LIN {X 0,Y 500.021,Z 595.129,A -85,B 0,C 180,E1 -13691.31,E2 -13691.31} C_VEL
LIN {X 0,Y 499.964,Z 595.135,A -85,B 0,C 180,E1 -13694.832,E2 -13694.832} C_VEL
LIN {X 0,Y 499.873,Z 595.155,A -85,B 0,C 180,E1 -13697.955,E2 -13697.955} C_VEL
LIN {X 0,Y 499.868,Z 595.149,A -85,B 0,C 180,E1 -13700.507,E2 -13700.507} C_VEL
LIN {X 0,Y 499.856,Z 595.149,A -85,B 0,C 180,E1 -13703.102,E2 -13703.102} C_VEL
LIN {X 0,Y 499.832,Z 595.157,A -85,B 0,C 180,E1 -13705.749,E2 -13705.749} C_VEL
LIN {X 0,Y 499.854,Z 595.151,A -85,B 0,C 180,E1 -13708.453,E2 -13708.453} C_VEL
LIN {X 0,Y 499.831,Z 595.152,A -85,B 0,C 180,E1 -13711.259,E2 -13711.259} C_VEL
LIN {X 0,Y 499.847,Z 595.155,A -85,B 0,C 180,E1 -13714.231,E2 -13714.231} C_VEL
LIN {X 0,Y 499.88,Z 595.146,A -85,B 0,C 180,E1 -13717.051,E2 -13717.051} C_VEL
LIN {X 0,Y 499.824,Z 595.159,A -85,B 0,C 180,E1 -13720.138,E2 -13720.138} C_VEL
LIN {X 0,Y 499.878,Z 595.147,A -85,B 0,C 180,E1 -13723.362,E2 -13723.362} C_VEL
LIN {X 0,Y 499.877,Z 595.146,A -85,B 0,C 180,E1 -13726.773,E2 -13726.773} C_VEL
LIN {X 0,Y 499.823,Z 595.16,A -85,B 0,C 180,E1 -13729.862,E2 -13729.862} C_VEL
LIN {X 0,Y 499.832,Z 595.151,A -85,B 0,C 180,E1 -13733.013,E2 -13733.013} C_VEL
LIN {X 0,Y 499.84,Z 595.158,A -85,B 0,C 180,E1 -13735.907,E2 -13735.907} C_VEL
LIN {X 0,Y 499.835,Z 595.152,A -85,B 0,C 180,E1 -13738.768,E2 -13738.768} C_VEL
LIN {X 0,Y 499.834,Z 595.154,A -85,B 0,C 180,E1 -13741.546,E2 -13741.546} C_VEL
LIN {X 0,Y 499.832,Z 595.16,A -85,B 0,C 180,E1 -13744.252,E2 -13744.252} C_VEL
LIN {X 0,Y 499.914,Z 595.236,A -85,B 0,C 180,E1 -13745.236,E2 -13745.236} C_VEL
LIN {X 0,Y 502.292,Z 608.896,A -85,B 0,C 180,E1 -13747.882,E2 -13747.882} C_VEL
LIN {X 0,Y 501.344,Z 623.933,A -85,B 0,C 180,E1 -13750.621,E2 -13750.621} C_VEL
LIN {X 0,Y 500.239,Z 642.384,A -85,B 0,C 180,E1 -13753.946,E2 -13753.946} C_VEL
LIN {X 0,Y 500.096,Z 646.425,A -85,B 0,C 180,E1 -13754.636,E2 -13754.636} C_VEL
LIN {X 0,Y 503.159,Z 673.816,A -85,B 0,C 180,E1 -13755.185,E2 -13755.185} C_VEL
LIN {X 0,Y 501.946,Z 752.433,A -85,B 0,C 180,E1 -13756.534,E2 -13756.534} C_VEL
LIN {X 0,Y 501.731,Z 762.36,A -85,B 0,C 180,E1 -13756.785,E2 -13756.785} C_VEL
LIN {X 0,Y 501.395,Z 772.419,A -85,B 0,C 180,E1 -13757.136,E2 -13757.136} C_VEL
LIN {X 0,Y 501.08,Z 782.406,A -85,B 0,C 180,E1 -13757.589,E2 -13757.589} C_VEL
LIN {X 0,Y 500.684,Z 792.552,A -85,B 0,C 180,E1 -13758.17,E2 -13758.17} C_VEL
LIN {X 0,Y 500.217,Z 802.826,A -85,B 0,C 180,E1 -13758.899,E2 -13758.899} C_VEL
LIN {X 0,Y 499.783,Z 811.123,A -85,B 0,C 180,E1 -13759.605,E2 -13759.605} C_VEL
LIN {X 0,Y 499.348,Z 820.005,A -85,B 0,C 180,E1 -13760.513,E2 -13760.513} C_VEL
LIN {X 0,Y 498.984,Z 826.725,A -85,B 0,C 180,E1 -13761.321,E2 -13761.321} C_VEL
LIN {X 0,Y 498.712,Z 833.772,A -85,B 0,C 180,E1 -13762.332,E2 -13762.332} C_VEL
LIN {X 0,Y 498.462,Z 840.635,A -85,B 0,C 180,E1 -13763.545,E2 -13763.545} C_VEL
LIN {X 0,Y 498.34,Z 844.527,A -85,B 0,C 180,E1 -13764.354,E2 -13764.354} C_VEL
LIN {X 0,Y 498.199,Z 849.173,A -85,B 0,C 180,E1 -13765.565,E2 -13765.565} C_VEL
LIN {X 0,Y 498.143,Z 852.679,A -85,B 0,C 180,E1 -13766.776,E2 -13766.776} C_VEL
LIN {X 0,Y 498.16,Z 855.649,A -85,B 0,C 180,E1 -13768.389,E2 -13768.389} C_VEL
LIN {X 0,Y 498.171,Z 856.61,A -85,B 0,C 180,E1 -13769.195,E2 -13769.195} C_VEL
LIN {X 0,Y 498.15,Z 857.003,A -85,B 0,C 180,E1 -13770.806,E2 -13770.806} C_VEL
LIN {X 0,Y 498.124,Z 856.638,A -85,B 0,C 180,E1 -13771.612,E2 -13771.612} C_VEL
LIN {X 0,Y 498.144,Z 854.362,A -85,B 0,C 180,E1 -13773.306,E2 -13773.306} C_VEL
LIN {X 0,Y 498.201,Z 851.826,A -85,B 0,C 180,E1 -13774.435,E2 -13774.435} C_VEL
LIN {X 0,Y 498.384,Z 848.053,A -85,B 0,C 180,E1 -13775.646,E2 -13775.646} C_VEL
LIN {X 0,Y 498.634,Z 843.12,A -85,B 0,C 180,E1 -13776.858,E2 -13776.858} C_VEL
LIN {X 0,Y 499.019,Z 836.872,A -85,B 0,C 180,E1 -13778.069,E2 -13778.069} C_VEL
LIN {X 0,Y 499.423,Z 830.563,A -85,B 0,C 180,E1 -13779.078,E2 -13779.078} C_VEL
LIN {X 0,Y 500.017,Z 822.995,A -85,B 0,C 180,E1 -13780.085,E2 -13780.085} C_VEL
LIN {X 0,Y 500.639,Z 814.859,A -85,B 0,C 180,E1 -13780.99,E2 -13780.99} C_VEL
LIN {X 0,Y 501.277,Z 805.922,A -85,B 0,C 180,E1 -13781.82,E2 -13781.82} C_VEL
LIN {X 0,Y 501.901,Z 796.264,A -85,B 0,C 180,E1 -13782.565,E2 -13782.565} C_VEL
LIN {X 0,Y 502.454,Z 786.303,A -85,B 0,C 180,E1 -13783.196,E2 -13783.196} C_VEL
LIN {X 0,Y 503.002,Z 776.582,A -85,B 0,C 180,E1 -13783.694,E2 -13783.694} C_VEL
LIN {X 0,Y 503.622,Z 765.279,A -85,B 0,C 180,E1 -13784.138,E2 -13784.138} C_VEL
LIN {X 0,Y 504.029,Z 755.185,A -85,B 0,C 180,E1 -13784.435,E2 -13784.435} C_VEL
LIN {X 0,Y 504.455,Z 737.22,A -85,B 0,C 180,E1 -13784.782,E2 -13784.782} C_VEL
LIN {X 0,Y 505.705,Z 672.59,A -85,B 0,C 180,E1 -13785.956,E2 -13785.956} C_VEL
LIN {X 0,Y 503.052,Z 654.485,A -85,B 0,C 180,E1 -13786.438,E2 -13786.438} C_VEL
LIN {X 0,Y 501.115,Z 644.89,A -85,B 0,C 180,E1 -13786.724,E2 -13786.724} C_VEL
LIN {X 0,Y 502.421,Z 628.877,A -85,B 0,C 180,E1 -13789.76,E2 -13789.76} C_VEL
LIN {X 0,Y 503.702,Z 615.998,A -85,B 0,C 180,E1 -13792.268,E2 -13792.268} C_VEL
LIN {X 0,Y 503.047,Z 610.412,A -85,B 0,C 180,E1 -13793.467,E2 -13793.467} C_VEL
LIN {X 0,Y 501.107,Z 600.725,A -85,B 0,C 180,E1 -13795.678,E2 -13795.678} C_VEL
LIN {X 0,Y 499.876,Z 595.157,A -85,B 0,C 180,E1 -13797.035,E2 -13797.035} C_VEL
LIN {X 0,Y 499.844,Z 595.157,A -85,B 0,C 180,E1 -13800.297,E2 -13800.297} C_VEL
LIN {X 0,Y 499.851,Z 595.156,A -85,B 0,C 180,E1 -13803.128,E2 -13803.128} C_VEL
LIN {X 0,Y 499.902,Z 595.145,A -85,B 0,C 180,E1 -13806.05,E2 -13806.05} C_VEL
LIN {X 0,Y 499.84,Z 595.151,A -85,B 0,C 180,E1 -13809.095,E2 -13809.095} C_VEL
LIN {X 0,Y 499.843,Z 595.15,A -85,B 0,C 180,E1 -13812.271,E2 -13812.271} C_VEL
LIN {X 0,Y 499.883,Z 595.148,A -85,B 0,C 180,E1 -13814.476,E2 -13814.476} C_VEL
LIN {X 0,Y 499.858,Z 595.154,A -85,B 0,C 180,E1 -13817.731,E2 -13817.731} C_VEL
LIN {X 0,Y 499.895,Z 595.148,A -85,B 0,C 180,E1 -13820.413,E2 -13820.413} C_VEL
LIN {X 0,Y 499.908,Z 595.145,A -85,B 0,C 180,E1 -13823.951,E2 -13823.951} C_VEL
LIN {X 0,Y 499.9,Z 595.149,A -85,B 0,C 180,E1 -13827.215,E2 -13827.215} C_VEL
LIN {X 0,Y 499.889,Z 595.148,A -85,B 0,C 180,E1 -13830.313,E2 -13830.313} C_VEL
LIN {X 0,Y 499.884,Z 595.151,A -85,B 0,C 180,E1 -13833.36,E2 -13833.36} C_VEL
LIN {X 0,Y 499.88,Z 595.15,A -85,B 0,C 180,E1 -13836.024,E2 -13836.024} C_VEL
LIN {X 0,Y 499.921,Z 595.151,A -85,B 0,C 180,E1 -13838.636,E2 -13838.636} C_VEL
LIN {X 0,Y 499.892,Z 595.155,A -85,B 0,C 180,E1 -13841.199,E2 -13841.199} C_VEL
LIN {X 0,Y 499.902,Z 595.151,A -85,B 0,C 180,E1 -13843.726,E2 -13843.726} C_VEL
LIN {X 0,Y 499.988,Z 595.223,A -85,B 0,C 180,E1 -13845.964,E2 -13845.964} C_VEL
LIN {X 0,Y 502.17,Z 605.861,A -85,B 0,C 180,E1 -13848.739,E2 -13848.739} C_VEL
LIN {X 0,Y 502.914,Z 610.897,A -85,B 0,C 180,E1 -13849.974,E2 -13849.974} C_VEL
LIN {X 0,Y 502.468,Z 618.166,A -85,B 0,C 180,E1 -13851.623,E2 -13851.623} C_VEL
LIN {X 0,Y 501.77,Z 626.142,A -85,B 0,C 180,E1 -13853.361,E2 -13853.361} C_VEL
LIN {X 0,Y 505.297,Z 642.925,A -85,B 0,C 180,E1 -13853.87,E2 -13853.87} C_VEL
LIN {X 0,Y 506.244,Z 649.346,A -85,B 0,C 180,E1 -13854.043,E2 -13854.043} C_VEL
LIN {X 0,Y 504.557,Z 711.904,A -85,B 0,C 180,E1 -13855.172,E2 -13855.172} C_VEL
LIN {X 0,Y 504.07,Z 733.839,A -85,B 0,C 180,E1 -13855.592,E2 -13855.592} C_VEL
LIN {X 0,Y 503.663,Z 745.565,A -85,B 0,C 180,E1 -13855.938,E2 -13855.938} C_VEL
LIN {X 0,Y 503.125,Z 759.1,A -85,B 0,C 180,E1 -13856.508,E2 -13856.508} C_VEL
LIN {X 0,Y 502.558,Z 771.102,A -85,B 0,C 180,E1 -13857.204,E2 -13857.204} C_VEL
LIN {X 0,Y 502.01,Z 780.801,A -85,B 0,C 180,E1 -13857.901,E2 -13857.901} C_VEL
LIN {X 0,Y 501.393,Z 789.985,A -85,B 0,C 180,E1 -13858.699,E2 -13858.699} C_VEL
LIN {X 0,Y 500.692,Z 798.607,A -85,B 0,C 180,E1 -13859.599,E2 -13859.599} C_VEL
LIN {X 0,Y 500.106,Z 805.153,A -85,B 0,C 180,E1 -13860.401,E2 -13860.401} C_VEL
LIN {X 0,Y 499.598,Z 812.014,A -85,B 0,C 180,E1 -13861.406,E2 -13861.406} C_VEL
LIN {X 0,Y 499.104,Z 817.772,A -85,B 0,C 180,E1 -13862.413,E2 -13862.413} C_VEL
LIN {X 0,Y 498.802,Z 823.337,A -85,B 0,C 180,E1 -13863.623,E2 -13863.623} C_VEL
LIN {X 0,Y 498.54,Z 827.721,A -85,B 0,C 180,E1 -13864.835,E2 -13864.835} C_VEL
LIN {X 0,Y 498.413,Z 830.206,A -85,B 0,C 180,E1 -13865.706,E2 -13865.706} C_VEL
LIN {X 0,Y 498.149,Z 833.293,A -85,B 0,C 180,E1 -13867.27,E2 -13867.27} C_VEL
LIN {X 0,Y 498.062,Z 834.271,A -85,B 0,C 180,E1 -13868.084,E2 -13868.084} C_VEL
LIN {X 0,Y 498.099,Z 834.913,A -85,B 0,C 180,E1 -13869.715,E2 -13869.715} C_VEL
LIN {X 0,Y 498.076,Z 834.546,A -85,B 0,C 180,E1 -13870.534,E2 -13870.534} C_VEL
LIN {X 0,Y 498.017,Z 832.61,A -85,B 0,C 180,E1 -13872.179,E2 -13872.179} C_VEL
LIN {X 0,Y 498.168,Z 829.923,A -85,B 0,C 180,E1 -13873.414,E2 -13873.414} C_VEL
LIN {X 0,Y 498.34,Z 826.113,A -85,B 0,C 180,E1 -13874.655,E2 -13874.655} C_VEL
LIN {X 0,Y 498.51,Z 821.045,A -85,B 0,C 180,E1 -13875.901,E2 -13875.901} C_VEL
LIN {X 0,Y 498.76,Z 815.812,A -85,B 0,C 180,E1 -13876.942,E2 -13876.942} C_VEL
LIN {X 0,Y 498.967,Z 809.412,A -85,B 0,C 180,E1 -13877.989,E2 -13877.989} C_VEL
LIN {X 0,Y 499.369,Z 801.644,A -85,B 0,C 180,E1 -13879.033,E2 -13879.033} C_VEL
LIN {X 0,Y 499.785,Z 792.659,A -85,B 0,C 180,E1 -13880.028,E2 -13880.028} C_VEL
LIN {X 0,Y 500.124,Z 784.129,A -85,B 0,C 180,E1 -13880.817,E2 -13880.817} C_VEL
LIN {X 0,Y 500.617,Z 774.605,A -85,B 0,C 180,E1 -13881.548,E2 -13881.548} C_VEL
LIN {X 0,Y 501.03,Z 764.623,A -85,B 0,C 180,E1 -13882.176,E2 -13882.176} C_VEL
LIN {X 0,Y 501.379,Z 754.57,A -85,B 0,C 180,E1 -13882.687,E2 -13882.687} C_VEL
LIN {X 0,Y 501.611,Z 743.432,A -85,B 0,C 180,E1 -13883.124,E2 -13883.124} C_VEL
LIN {X 0,Y 501.903,Z 732.354,A -85,B 0,C 180,E1 -13883.437,E2 -13883.437} C_VEL
LIN {X 0,Y 502.427,Z 709.429,A -85,B 0,C 180,E1 -13883.847,E2 -13883.847} C_VEL
LIN {X 0,Y 503.284,Z 645.821,A -85,B 0,C 180,E1 -13884.934,E2 -13884.934} C_VEL
LIN {X 0,Y 500.222,Z 624.306,A -85,B 0,C 180,E1 -13885.398,E2 -13885.398} C_VEL
LIN {X 0,Y 501.029,Z 609.69,A -85,B 0,C 180,E1 -13888.38,E2 -13888.38} C_VEL
LIN {X 0,Y 501.279,Z 603.782,A -85,B 0,C 180,E1 -13889.603,E2 -13889.603} C_VEL
LIN {X 0,Y 499.955,Z 595.145,A -85,B 0,C 180,E1 -13891.488,E2 -13891.488} C_VEL
LIN {X 0,Y 499.881,Z 595.15,A -85,B 0,C 180,E1 -13894.236,E2 -13894.236} C_VEL
LIN {X 0,Y 499.889,Z 595.144,A -85,B 0,C 180,E1 -13897.05,E2 -13897.05} C_VEL
LIN {X 0,Y 499.879,Z 595.152,A -85,B 0,C 180,E1 -13900.132,E2 -13900.132} C_VEL
LIN {X 0,Y 499.88,Z 595.147,A -85,B 0,C 180,E1 -13903.361,E2 -13903.361} C_VEL
LIN {X 0,Y 499.88,Z 595.146,A -85,B 0,C 180,E1 -13906.638,E2 -13906.638} C_VEL
LIN {X 0,Y 499.878,Z 595.153,A -85,B 0,C 180,E1 -13909.867,E2 -13909.867} C_VEL
LIN {X 0,Y 499.89,Z 595.144,A -85,B 0,C 180,E1 -13913.004,E2 -13913.004} C_VEL
LIN {X 0,Y 499.869,Z 595.155,A -85,B 0,C 180,E1 -13915.909,E2 -13915.909} C_VEL
LIN {X 0,Y 499.875,Z 595.147,A -85,B 0,C 180,E1 -13918.771,E2 -13918.771} C_VEL
LIN {X 0,Y 499.898,Z 595.152,A -85,B 0,C 180,E1 -13921.974,E2 -13921.974} C_VEL
LIN {X 0,Y 499.837,Z 595.156,A -85,B 0,C 180,E1 -13924.252,E2 -13924.252} C_VEL
LIN {X 0,Y 499.857,Z 595.148,A -85,B 0,C 180,E1 -13926.898,E2 -13926.898} C_VEL
LIN {X 0,Y 499.917,Z 595.148,A -85,B 0,C 180,E1 -13929.841,E2 -13929.841} C_VEL
LIN {X 0,Y 499.916,Z 595.141,A -85,B 0,C 180,E1 -13932.888,E2 -13932.888} C_VEL
LIN {X 0,Y 499.993,Z 595.133,A -85,B 0,C 180,E1 -13935.394,E2 -13935.394} C_VEL
LIN {X 0,Y 500.036,Z 595.127,A -85,B 0,C 180,E1 -13938.69,E2 -13938.69} C_VEL
LIN {X 0,Y 500.029,Z 595.135,A -85,B 0,C 180,E1 -13941.947,E2 -13941.947} C_VEL
LIN {X 0,Y 500.166,Z 595.11,A -85,B 0,C 180,E1 -13945.18,E2 -13945.18} C_VEL
LIN {X 0,Y 500.148,Z 595.112,A -85,B 0,C 180,E1 -13949.197,E2 -13949.197} C_VEL
LIN {X 0,Y 500.148,Z 595.112,A -85,B 0,C 180,E1 -13950.802,E2 -13950.802} C_VEL
LIN {X 0,Y 500.165,Z 595.11,A -85,B 0,C 180,E1 -13954.82,E2 -13954.82} C_VEL
LIN {X 0,Y 500.029,Z 595.135,A -85,B 0,C 180,E1 -13958.052,E2 -13958.052} C_VEL
LIN {X 0,Y 499.959,Z 595.137,A -85,B 0,C 180,E1 -13960.087,E2 -13960.087} C_VEL
LIN {X 0,Y 499.321,Z 595.218,A -85,B 0,C 180,E1 -13960.76,E2 -13960.76} C_VEL
LIN {X 0,Y 496.455,Z 595.579,A -85,B 0,C 180,E1 -13961.851,E2 -13961.851} C_VEL
LIN {X 0,Y 494.018,Z 595.878,A -85,B 0,C 180,E1 -13962.731,E2 -13962.731} C_VEL
LIN {X 0,Y 492.979,Z 596.007,A -85,B 0,C 180,E1 -13963.411,E2 -13963.411} C_VEL
LIN {X 0,Y 492.901,Z 596.019,A -85,B 0,C 180,E1 -13963.642,E2 -13963.642} C_VEL
LIN {X 0,Y 492.898,Z 596.019,A -85,B 0,C 180,E1 -13965.664,E2 -13965.664} C_VEL
LIN {X 0,Y 492.876,Z 596.023,A -85,B 0,C 180,E1 -13968.219,E2 -13968.219} C_VEL
LIN {X 0,Y 492.862,Z 596.02,A -85,B 0,C 180,E1 -13970.811,E2 -13970.811} C_VEL
LIN {X 0,Y 492.813,Z 596.028,A -85,B 0,C 180,E1 -13973.451,E2 -13973.451} C_VEL
LIN {X 0,Y 492.84,Z 596.025,A -85,B 0,C 180,E1 -13976.444,E2 -13976.444} C_VEL
LIN {X 0,Y 492.831,Z 596.024,A -85,B 0,C 180,E1 -13978.896,E2 -13978.896} C_VEL
LIN {X 0,Y 492.857,Z 596.025,A -85,B 0,C 180,E1 -13981.725,E2 -13981.725} C_VEL
LIN {X 0,Y 492.852,Z 596.022,A -85,B 0,C 180,E1 -13984.644,E2 -13984.644} C_VEL
LIN {X 0,Y 492.858,Z 596.024,A -85,B 0,C 180,E1 -13987.67,E2 -13987.67} C_VEL
LIN {X 0,Y 492.846,Z 596.022,A -85,B 0,C 180,E1 -13990.826,E2 -13990.826} C_VEL
LIN {X 0,Y 492.835,Z 596.029,A -85,B 0,C 180,E1 -13994.14,E2 -13994.14} C_VEL
LIN {X 0,Y 492.839,Z 596.023,A -85,B 0,C 180,E1 -13996.985,E2 -13996.985} C_VEL
LIN {X 0,Y 492.857,Z 596.025,A -85,B 0,C 180,E1 -14000.243,E2 -14000.243} C_VEL
LIN {X 0,Y 492.86,Z 596.021,A -85,B 0,C 180,E1 -14003.353,E2 -14003.353} C_VEL
LIN {X 0,Y 492.819,Z 596.029,A -85,B 0,C 180,E1 -14006.337,E2 -14006.337} C_VEL
LIN {X 0,Y 492.82,Z 596.025,A -85,B 0,C 180,E1 -14009.226,E2 -14009.226} C_VEL
LIN {X 0,Y 492.864,Z 596.027,A -85,B 0,C 180,E1 -14012.032,E2 -14012.032} C_VEL
LIN {X 0,Y 492.785,Z 596.03,A -85,B 0,C 180,E1 -14014.76,E2 -14014.76} C_VEL
LIN {X 0,Y 492.858,Z 596.022,A -85,B 0,C 180,E1 -14017.484,E2 -14017.484} C_VEL
LIN {X 0,Y 492.882,Z 596.025,A -85,B 0,C 180,E1 -14020.058,E2 -14020.058} C_VEL
LIN {X 0,Y 492.87,Z 596.02,A -85,B 0,C 180,E1 -14022.636,E2 -14022.636} C_VEL
LIN {X 0,Y 492.933,Z 596.011,A -85,B 0,C 180,E1 -14025.181,E2 -14025.181} C_VEL
LIN {X 0,Y 493.001,Z 596.004,A -85,B 0,C 180,E1 -14028.618,E2 -14028.618} C_VEL
LIN {X 0,Y 492.978,Z 596.012,A -85,B 0,C 180,E1 -14031.832,E2 -14031.832} C_VEL
LIN {X 0,Y 493.053,Z 596,A -85,B 0,C 180,E1 -14034.293,E2 -14034.293} C_VEL
LIN {X 0,Y 492.992,Z 596.004,A -85,B 0,C 180,E1 -14036.742,E2 -14036.742} C_VEL
LIN {X 0,Y 493.182,Z 595.988,A -85,B 0,C 180,E1 -14040,E2 -14040} C_VEL
LIN {X 0,Y 493.064,Z 596.002,A -85,B 0,C 180,E1 -14044.073,E2 -14044.073} C_VEL
LIN {X 0,Y 493.031,Z 596.001,A -85,B 0,C 180,E1 -14046.526,E2 -14046.526} C_VEL
LIN {X 0,Y 492.95,Z 596.009,A -85,B 0,C 180,E1 -14048.993,E2 -14048.993} C_VEL
LIN {X 0,Y 492.973,Z 596.008,A -85,B 0,C 180,E1 -14051.474,E2 -14051.474} C_VEL
LIN {X 0,Y 492.912,Z 596.014,A -85,B 0,C 180,E1 -14054.917,E2 -14054.917} C_VEL
LIN {X 0,Y 492.828,Z 596.029,A -85,B 0,C 180,E1 -14058.221,E2 -14058.221} C_VEL
LIN {X 0,Y 492.83,Z 596.024,A -85,B 0,C 180,E1 -14060.813,E2 -14060.813} C_VEL
LIN {X 0,Y 492.814,Z 596.028,A -85,B 0,C 180,E1 -14063.451,E2 -14063.451} C_VEL
LIN {X 0,Y 492.82,Z 596.028,A -85,B 0,C 180,E1 -14066.438,E2 -14066.438} C_VEL
LIN {X 0,Y 492.831,Z 596.024,A -85,B 0,C 180,E1 -14068.897,E2 -14068.897} C_VEL
LIN {X 0,Y 492.767,Z 596.037,A -85,B 0,C 180,E1 -14071.731,E2 -14071.731} C_VEL
LIN {X 0,Y 492.813,Z 596.027,A -85,B 0,C 180,E1 -14074.648,E2 -14074.648} C_VEL
LIN {X 0,Y 492.789,Z 596.033,A -85,B 0,C 180,E1 -14077.676,E2 -14077.676} C_VEL
LIN {X 0,Y 492.771,Z 596.031,A -85,B 0,C 180,E1 -14080.834,E2 -14080.834} C_VEL
LIN {X 0,Y 492.832,Z 596.026,A -85,B 0,C 180,E1 -14083.544,E2 -14083.544} C_VEL
LIN {X 0,Y 492.832,Z 596.026,A -85,B 0,C 180,E1 -14086.456,E2 -14086.456} C_VEL
LIN {X 0,Y 492.77,Z 596.031,A -85,B 0,C 180,E1 -14089.167,E2 -14089.167} C_VEL
LIN {X 0,Y 492.752,Z 596.037,A -85,B 0,C 180,E1 -14092.321,E2 -14092.321} C_VEL
LIN {X 0,Y 492.812,Z 596.029,A -85,B 0,C 180,E1 -14095.524,E2 -14095.524} C_VEL
LIN {X 0,Y 492.773,Z 596.033,A -85,B 0,C 180,E1 -14098.524,E2 -14098.524} C_VEL
LIN {X 0,Y 492.82,Z 596.025,A -85,B 0,C 180,E1 -14101.103,E2 -14101.103} C_VEL
LIN {X 0,Y 492.817,Z 596.032,A -85,B 0,C 180,E1 -14103.858,E2 -14103.858} C_VEL
LIN {X 0,Y 492.844,Z 596.116,A -85,B 0,C 180,E1 -14105.118,E2 -14105.118} C_VEL
LIN {X 0,Y 495.229,Z 609.593,A -85,B 0,C 180,E1 -14107.769,E2 -14107.769} C_VEL
LIN {X 0,Y 494.467,Z 622.315,A -85,B 0,C 180,E1 -14110.125,E2 -14110.125} C_VEL
LIN {X 0,Y 493.253,Z 641.911,A -85,B 0,C 180,E1 -14113.712,E2 -14113.712} C_VEL
LIN {X 0,Y 493.06,Z 646.332,A -85,B 0,C 180,E1 -14114.474,E2 -14114.474} C_VEL
LIN {X 0,Y 496.152,Z 674.763,A -85,B 0,C 180,E1 -14115.054,E2 -14115.054} C_VEL
LIN {X 0,Y 494.92,Z 752.307,A -85,B 0,C 180,E1 -14116.418,E2 -14116.418} C_VEL
LIN {X 0,Y 494.724,Z 762.206,A -85,B 0,C 180,E1 -14116.673,E2 -14116.673} C_VEL
LIN {X 0,Y 494.35,Z 772.836,A -85,B 0,C 180,E1 -14117.053,E2 -14117.053} C_VEL
LIN {X 0,Y 494.025,Z 782.692,A -85,B 0,C 180,E1 -14117.513,E2 -14117.513} C_VEL
LIN {X 0,Y 493.648,Z 792.056,A -85,B 0,C 180,E1 -14118.054,E2 -14118.054} C_VEL
LIN {X 0,Y 493.201,Z 801.722,A -85,B 0,C 180,E1 -14118.739,E2 -14118.739} C_VEL
LIN {X 0,Y 492.71,Z 811.215,A -85,B 0,C 180,E1 -14119.557,E2 -14119.557} C_VEL
LIN {X 0,Y 492.33,Z 819.196,A -85,B 0,C 180,E1 -14120.377,E2 -14120.377} C_VEL
LIN {X 0,Y 491.866,Z 827.475,A -85,B 0,C 180,E1 -14121.401,E2 -14121.401} C_VEL
LIN {X 0,Y 491.597,Z 834.372,A -85,B 0,C 180,E1 -14122.427,E2 -14122.427} C_VEL
LIN {X 0,Y 491.365,Z 840.117,A -85,B 0,C 180,E1 -14123.452,E2 -14123.452} C_VEL
LIN {X 0,Y 491.261,Z 844.047,A -85,B 0,C 180,E1 -14124.272,E2 -14124.272} C_VEL
LIN {X 0,Y 491.115,Z 848.778,A -85,B 0,C 180,E1 -14125.501,E2 -14125.501} C_VEL
LIN {X 0,Y 491.072,Z 852.536,A -85,B 0,C 180,E1 -14126.808,E2 -14126.808} C_VEL
LIN {X 0,Y 491.062,Z 855.403,A -85,B 0,C 180,E1 -14128.365,E2 -14128.365} C_VEL
LIN {X 0,Y 491.087,Z 856.381,A -85,B 0,C 180,E1 -14129.183,E2 -14129.183} C_VEL
LIN {X 0,Y 491.067,Z 856.862,A -85,B 0,C 180,E1 -14130.817,E2 -14130.817} C_VEL
LIN {X 0,Y 491.028,Z 856.495,A -85,B 0,C 180,E1 -14131.635,E2 -14131.635} C_VEL
LIN {X 0,Y 491.07,Z 854.482,A -85,B 0,C 180,E1 -14133.271,E2 -14133.271} C_VEL
LIN {X 0,Y 491.118,Z 851.815,A -85,B 0,C 180,E1 -14134.499,E2 -14134.499} C_VEL
LIN {X 0,Y 491.327,Z 848.089,A -85,B 0,C 180,E1 -14135.727,E2 -14135.727} C_VEL
LIN {X 0,Y 491.567,Z 843.224,A -85,B 0,C 180,E1 -14136.957,E2 -14136.957} C_VEL
LIN {X 0,Y 491.991,Z 837.061,A -85,B 0,C 180,E1 -14138.185,E2 -14138.185} C_VEL
LIN {X 0,Y 492.429,Z 830.836,A -85,B 0,C 180,E1 -14139.208,E2 -14139.208} C_VEL
LIN {X 0,Y 493.044,Z 823.343,A -85,B 0,C 180,E1 -14140.229,E2 -14140.229} C_VEL
LIN {X 0,Y 493.753,Z 814.267,A -85,B 0,C 180,E1 -14141.248,E2 -14141.248} C_VEL
LIN {X 0,Y 494.371,Z 806.466,A -85,B 0,C 180,E1 -14141.988,E2 -14141.988} C_VEL
LIN {X 0,Y 495.047,Z 796.503,A -85,B 0,C 180,E1 -14142.773,E2 -14142.773} C_VEL
LIN {X 0,Y 495.587,Z 787.184,A -85,B 0,C 180,E1 -14143.382,E2 -14143.382} C_VEL
LIN {X 0,Y 496.224,Z 776.584,A -85,B 0,C 180,E1 -14143.937,E2 -14143.937} C_VEL
LIN {X 0,Y 496.861,Z 765.366,A -85,B 0,C 180,E1 -14144.387,E2 -14144.387} C_VEL
LIN {X 0,Y 497.342,Z 754.316,A -85,B 0,C 180,E1 -14144.711,E2 -14144.711} C_VEL
LIN {X 0,Y 497.891,Z 732.5,A -85,B 0,C 180,E1 -14145.138,E2 -14145.138} C_VEL
LIN {X 0,Y 499.162,Z 673.768,A -85,B 0,C 180,E1 -14146.235,E2 -14146.235} C_VEL
LIN {X 0,Y 496.551,Z 655.972,A -85,B 0,C 180,E1 -14146.719,E2 -14146.719} C_VEL
LIN {X 0,Y 494.29,Z 644.579,A -85,B 0,C 180,E1 -14147.09,E2 -14147.09} C_VEL
LIN {X 0,Y 495.715,Z 628.246,A -85,B 0,C 180,E1 -14150.254,E2 -14150.254} C_VEL
LIN {X 0,Y 496.835,Z 616.545,A -85,B 0,C 180,E1 -14152.593,E2 -14152.593} C_VEL
LIN {X 0,Y 495.331,Z 607.413,A -85,B 0,C 180,E1 -14154.645,E2 -14154.645} C_VEL
LIN {X 0,Y 493.181,Z 597.556,A -85,B 0,C 180,E1 -14157.032,E2 -14157.032} C_VEL
LIN {X 0,Y 492.813,Z 596.039,A -85,B 0,C 180,E1 -14157.454,E2 -14157.454} C_VEL
LIN {X 0,Y 492.817,Z 596.036,A -85,B 0,C 180,E1 -14159.889,E2 -14159.889} C_VEL
LIN {X 0,Y 492.8,Z 596.034,A -85,B 0,C 180,E1 -14163.008,E2 -14163.008} C_VEL
LIN {X 0,Y 492.867,Z 596.022,A -85,B 0,C 180,E1 -14165.898,E2 -14165.898} C_VEL
LIN {X 0,Y 492.813,Z 596.023,A -85,B 0,C 180,E1 -14168.71,E2 -14168.71} C_VEL
LIN {X 0,Y 492.821,Z 596.025,A -85,B 0,C 180,E1 -14172.347,E2 -14172.347} C_VEL
LIN {X 0,Y 492.843,Z 596.026,A -85,B 0,C 180,E1 -14175.285,E2 -14175.285} C_VEL
LIN {X 0,Y 492.825,Z 596.029,A -85,B 0,C 180,E1 -14178.087,E2 -14178.087} C_VEL
LIN {X 0,Y 492.826,Z 596.03,A -85,B 0,C 180,E1 -14181.291,E2 -14181.291} C_VEL
LIN {X 0,Y 492.85,Z 596.025,A -85,B 0,C 180,E1 -14184.359,E2 -14184.359} C_VEL
LIN {X 0,Y 492.853,Z 596.026,A -85,B 0,C 180,E1 -14187.312,E2 -14187.312} C_VEL
LIN {X 0,Y 492.834,Z 596.026,A -85,B 0,C 180,E1 -14190.169,E2 -14190.169} C_VEL
LIN {X 0,Y 492.842,Z 596.028,A -85,B 0,C 180,E1 -14192.948,E2 -14192.948} C_VEL
LIN {X 0,Y 492.86,Z 596.024,A -85,B 0,C 180,E1 -14195.66,E2 -14195.66} C_VEL
LIN {X 0,Y 492.864,Z 596.03,A -85,B 0,C 180,E1 -14198.315,E2 -14198.315} C_VEL
LIN {X 0,Y 492.858,Z 596.033,A -85,B 0,C 180,E1 -14200.921,E2 -14200.921} C_VEL
LIN {X 0,Y 492.861,Z 596.027,A -85,B 0,C 180,E1 -14203.487,E2 -14203.487} C_VEL
LIN {X 0,Y 492.978,Z 596.209,A -85,B 0,C 180,E1 -14205.602,E2 -14205.602} C_VEL
LIN {X 0,Y 495,Z 606.134,A -85,B 0,C 180,E1 -14208.268,E2 -14208.268} C_VEL
LIN {X 0,Y 496.017,Z 612.283,A -85,B 0,C 180,E1 -14209.833,E2 -14209.833} C_VEL
LIN {X 0,Y 495.606,Z 619.545,A -85,B 0,C 180,E1 -14211.507,E2 -14211.507} C_VEL
LIN {X 0,Y 494.995,Z 626.457,A -85,B 0,C 180,E1 -14213.028,E2 -14213.028} C_VEL
LIN {X 0,Y 498.807,Z 644.301,A -85,B 0,C 180,E1 -14213.588,E2 -14213.588} C_VEL
LIN {X 0,Y 499.675,Z 649.606,A -85,B 0,C 180,E1 -14213.738,E2 -14213.738} C_VEL
LIN {X 0,Y 497.89,Z 712.846,A -85,B 0,C 180,E1 -14214.905,E2 -14214.905} C_VEL
LIN {X 0,Y 497.334,Z 735.301,A -85,B 0,C 180,E1 -14215.355,E2 -14215.355} C_VEL
LIN {X 0,Y 496.789,Z 749.201,A -85,B 0,C 180,E1 -14215.805,E2 -14215.805} C_VEL
LIN {X 0,Y 496.261,Z 761.047,A -85,B 0,C 180,E1 -14216.358,E2 -14216.358} C_VEL
LIN {X 0,Y 495.774,Z 771.247,A -85,B 0,C 180,E1 -14216.963,E2 -14216.963} C_VEL
LIN {X 0,Y 495.2,Z 780.956,A -85,B 0,C 180,E1 -14217.669,E2 -14217.669} C_VEL
LIN {X 0,Y 494.518,Z 790.162,A -85,B 0,C 180,E1 -14218.478,E2 -14218.478} C_VEL
LIN {X 0,Y 493.975,Z 797.082,A -85,B 0,C 180,E1 -14219.187,E2 -14219.187} C_VEL
LIN {X 0,Y 493.185,Z 805.344,A -85,B 0,C 180,E1 -14220.203,E2 -14220.203} C_VEL
LIN {X 0,Y 492.624,Z 812.216,A -85,B 0,C 180,E1 -14221.222,E2 -14221.222} C_VEL
LIN {X 0,Y 492.149,Z 817.97,A -85,B 0,C 180,E1 -14222.243,E2 -14222.243} C_VEL
LIN {X 0,Y 491.752,Z 823.871,A -85,B 0,C 180,E1 -14223.561,E2 -14223.561} C_VEL
LIN {X 0,Y 491.58,Z 827.176,A -85,B 0,C 180,E1 -14224.454,E2 -14224.454} C_VEL
LIN {X 0,Y 491.335,Z 830.765,A -85,B 0,C 180,E1 -14225.727,E2 -14225.727} C_VEL
LIN {X 0,Y 491.037,Z 833.706,A -85,B 0,C 180,E1 -14227.376,E2 -14227.376} C_VEL
LIN {X 0,Y 490.985,Z 834.654,A -85,B 0,C 180,E1 -14228.202,E2 -14228.202} C_VEL
LIN {X 0,Y 491.002,Z 834.991,A -85,B 0,C 180,E1 -14229.857,E2 -14229.857} C_VEL
LIN {X 0,Y 490.974,Z 834.616,A -85,B 0,C 180,E1 -14230.688,E2 -14230.688} C_VEL
LIN {X 0,Y 490.932,Z 832.335,A -85,B 0,C 180,E1 -14232.357,E2 -14232.357} C_VEL
LIN {X 0,Y 491.114,Z 829.456,A -85,B 0,C 180,E1 -14233.611,E2 -14233.611} C_VEL
LIN {X 0,Y 491.259,Z 825.433,A -85,B 0,C 180,E1 -14234.871,E2 -14234.871} C_VEL
LIN {X 0,Y 491.428,Z 821.157,A -85,B 0,C 180,E1 -14235.924,E2 -14235.924} C_VEL
LIN {X 0,Y 491.679,Z 815.946,A -85,B 0,C 180,E1 -14236.972,E2 -14236.972} C_VEL
LIN {X 0,Y 491.896,Z 809.479,A -85,B 0,C 180,E1 -14238.042,E2 -14238.042} C_VEL
LIN {X 0,Y 492.293,Z 801.679,A -85,B 0,C 180,E1 -14239.101,E2 -14239.101} C_VEL
LIN {X 0,Y 492.722,Z 793.232,A -85,B 0,C 180,E1 -14240.054,E2 -14240.054} C_VEL
LIN {X 0,Y 493.072,Z 784.093,A -85,B 0,C 180,E1 -14240.911,E2 -14240.911} C_VEL
LIN {X 0,Y 493.566,Z 774.519,A -85,B 0,C 180,E1 -14241.652,E2 -14241.652} C_VEL
LIN {X 0,Y 494.008,Z 764.489,A -85,B 0,C 180,E1 -14242.289,E2 -14242.289} C_VEL
LIN {X 0,Y 494.371,Z 754.361,A -85,B 0,C 180,E1 -14242.807,E2 -14242.807} C_VEL
LIN {X 0,Y 494.597,Z 743.547,A -85,B 0,C 180,E1 -14243.236,E2 -14243.236} C_VEL
LIN {X 0,Y 494.877,Z 733.045,A -85,B 0,C 180,E1 -14243.541,E2 -14243.541} C_VEL
LIN {X 0,Y 495.296,Z 713.357,A -85,B 0,C 180,E1 -14243.907,E2 -14243.907} C_VEL
LIN {X 0,Y 496.342,Z 646.943,A -85,B 0,C 180,E1 -14245.067,E2 -14245.067} C_VEL
LIN {X 0,Y 493.234,Z 624.467,A -85,B 0,C 180,E1 -14245.555,E2 -14245.555} C_VEL
LIN {X 0,Y 494.011,Z 610.385,A -85,B 0,C 180,E1 -14248.468,E2 -14248.468} C_VEL
LIN {X 0,Y 494.239,Z 604.332,A -85,B 0,C 180,E1 -14249.737,E2 -14249.737} C_VEL
LIN {X 0,Y 492.895,Z 596.024,A -85,B 0,C 180,E1 -14251.574,E2 -14251.574} C_VEL
LIN {X 0,Y 492.837,Z 596.024,A -85,B 0,C 180,E1 -14254.645,E2 -14254.645} C_VEL
LIN {X 0,Y 492.844,Z 596.023,A -85,B 0,C 180,E1 -14257.26,E2 -14257.26} C_VEL
LIN {X 0,Y 492.835,Z 596.03,A -85,B 0,C 180,E1 -14259.872,E2 -14259.872} C_VEL
LIN {X 0,Y 492.841,Z 596.022,A -85,B 0,C 180,E1 -14263.015,E2 -14263.015} C_VEL
LIN {X 0,Y 492.837,Z 596.03,A -85,B 0,C 180,E1 -14265.86,E2 -14265.86} C_VEL
LIN {X 0,Y 492.847,Z 596.022,A -85,B 0,C 180,E1 -14269.174,E2 -14269.174} C_VEL
LIN {X 0,Y 492.797,Z 596.032,A -85,B 0,C 180,E1 -14272.324,E2 -14272.324} C_VEL
LIN {X 0,Y 492.845,Z 596.025,A -85,B 0,C 180,E1 -14274.359,E2 -14274.359} C_VEL
LIN {X 0,Y 492.801,Z 596.028,A -85,B 0,C 180,E1 -14277.308,E2 -14277.308} C_VEL
LIN {X 0,Y 492.826,Z 596.03,A -85,B 0,C 180,E1 -14280.168,E2 -14280.168} C_VEL
LIN {X 0,Y 492.838,Z 596.023,A -85,B 0,C 180,E1 -14282.948,E2 -14282.948} C_VEL
LIN {X 0,Y 492.854,Z 596.025,A -85,B 0,C 180,E1 -14285.66,E2 -14285.66} C_VEL
LIN {X 0,Y 492.858,Z 596.024,A -85,B 0,C 180,E1 -14288.314,E2 -14288.314} C_VEL
LIN {X 0,Y 492.853,Z 596.021,A -85,B 0,C 180,E1 -14290.92,E2 -14290.92} C_VEL
LIN {X 0,Y 492.868,Z 596.021,A -85,B 0,C 180,E1 -14293.487,E2 -14293.487} C_VEL
LIN {X 0,Y 492.916,Z 596.021,A -85,B 0,C 180,E1 -14296.02,E2 -14296.02} C_VEL
LIN {X 0,Y 492.971,Z 596.007,A -85,B 0,C 180,E1 -14299.355,E2 -14299.355} C_VEL
LIN {X 0,Y 493.009,Z 596.002,A -85,B 0,C 180,E1 -14302.653,E2 -14302.653} C_VEL
LIN {X 0,Y 493.116,Z 595.988,A -85,B 0,C 180,E1 -14305.111,E2 -14305.111} C_VEL
LIN {X 0,Y 493.098,Z 595.991,A -85,B 0,C 180,E1 -14309.186,E2 -14309.186} C_VEL
LIN {X 0,Y 493.098,Z 595.991,A -85,B 0,C 180,E1 -14310.814,E2 -14310.814} C_VEL
LIN {X 0,Y 493.116,Z 595.988,A -85,B 0,C 180,E1 -14314.889,E2 -14314.889} C_VEL
LIN {X 0,Y 492.973,Z 596.012,A -85,B 0,C 180,E1 -14318.168,E2 -14318.168} C_VEL
LIN {X 0,Y 492.969,Z 596.008,A -85,B 0,C 180,E1 -14321.474,E2 -14321.474} C_VEL
LIN {X 0,Y 492.901,Z 596.019,A -85,B 0,C 180,E1 -14323.642,E2 -14323.642} C_VEL
LIN {X 0,Y 492.239,Z 596.106,A -85,B 0,C 180,E1 -14324.324,E2 -14324.324} C_VEL
LIN {X 0,Y 489.352,Z 596.463,A -85,B 0,C 180,E1 -14325.432,E2 -14325.432} C_VEL
LIN {X 0,Y 486.919,Z 596.764,A -85,B 0,C 180,E1 -14326.324,E2 -14326.324} C_VEL
LIN {X 0,Y 485.896,Z 596.888,A -85,B 0,C 180,E1 -14327.014,E2 -14327.014} C_VEL
LIN {X 0,Y 485.825,Z 596.897,A -85,B 0,C 180,E1 -14327.248,E2 -14327.248} C_VEL
LIN {X 0,Y 485.82,Z 596.9,A -85,B 0,C 180,E1 -14330.422,E2 -14330.422} C_VEL
LIN {X 0,Y 485.78,Z 596.902,A -85,B 0,C 180,E1 -14332.912,E2 -14332.912} C_VEL
LIN {X 0,Y 485.766,Z 596.907,A -85,B 0,C 180,E1 -14335.631,E2 -14335.631} C_VEL
LIN {X 0,Y 485.801,Z 596.902,A -85,B 0,C 180,E1 -14338.417,E2 -14338.417} C_VEL
LIN {X 0,Y 485.812,Z 596.903,A -85,B 0,C 180,E1 -14341.717,E2 -14341.717} C_VEL
LIN {X 0,Y 485.802,Z 596.9,A -85,B 0,C 180,E1 -14344.731,E2 -14344.731} C_VEL
LIN {X 0,Y 485.817,Z 596.9,A -85,B 0,C 180,E1 -14347.536,E2 -14347.536} C_VEL
LIN {X 0,Y 485.791,Z 596.903,A -85,B 0,C 180,E1 -14350.454,E2 -14350.454} C_VEL
LIN {X 0,Y 485.784,Z 596.908,A -85,B 0,C 180,E1 -14353.868,E2 -14353.868} C_VEL
LIN {X 0,Y 485.786,Z 596.906,A -85,B 0,C 180,E1 -14356.204,E2 -14356.204} C_VEL
LIN {X 0,Y 485.792,Z 596.903,A -85,B 0,C 180,E1 -14359.547,E2 -14359.547} C_VEL
LIN {X 0,Y 485.831,Z 596.896,A -85,B 0,C 180,E1 -14362.733,E2 -14362.733} C_VEL
LIN {X 0,Y 485.798,Z 596.905,A -85,B 0,C 180,E1 -14365.784,E2 -14365.784} C_VEL
LIN {X 0,Y 485.783,Z 596.902,A -85,B 0,C 180,E1 -14368.73,E2 -14368.73} C_VEL
LIN {X 0,Y 485.802,Z 596.902,A -85,B 0,C 180,E1 -14371.589,E2 -14371.589} C_VEL
LIN {X 0,Y 485.771,Z 596.906,A -85,B 0,C 180,E1 -14374.369,E2 -14374.369} C_VEL
LIN {X 0,Y 485.786,Z 596.902,A -85,B 0,C 180,E1 -14377.339,E2 -14377.339} C_VEL
LIN {X 0,Y 485.843,Z 596.899,A -85,B 0,C 180,E1 -14379.757,E2 -14379.757} C_VEL
LIN {X 0,Y 485.84,Z 596.898,A -85,B 0,C 180,E1 -14382.377,E2 -14382.377} C_VEL
LIN {X 0,Y 485.872,Z 596.897,A -85,B 0,C 180,E1 -14385.814,E2 -14385.814} C_VEL
LIN {X 0,Y 485.956,Z 596.88,A -85,B 0,C 180,E1 -14389.2,E2 -14389.2} C_VEL
LIN {X 0,Y 485.963,Z 596.881,A -85,B 0,C 180,E1 -14392.547,E2 -14392.547} C_VEL
LIN {X 0,Y 486.041,Z 596.875,A -85,B 0,C 180,E1 -14394.211,E2 -14394.211} C_VEL
LIN {X 0,Y 485.973,Z 596.879,A -85,B 0,C 180,E1 -14396.695,E2 -14396.695} C_VEL
LIN {X 0,Y 486.136,Z 596.866,A -85,B 0,C 180,E1 -14400,E2 -14400} C_VEL
LIN {X 0,Y 486.027,Z 596.877,A -85,B 0,C 180,E1 -14404.132,E2 -14404.132} C_VEL
LIN {X 0,Y 485.991,Z 596.877,A -85,B 0,C 180,E1 -14406.621,E2 -14406.621} C_VEL
LIN {X 0,Y 485.919,Z 596.885,A -85,B 0,C 180,E1 -14409.124,E2 -14409.124} C_VEL
LIN {X 0,Y 485.913,Z 596.889,A -85,B 0,C 180,E1 -14411.643,E2 -14411.643} C_VEL
LIN {X 0,Y 485.868,Z 596.891,A -85,B 0,C 180,E1 -14415.04,E2 -14415.04} C_VEL
LIN {X 0,Y 485.791,Z 596.903,A -85,B 0,C 180,E1 -14418.494,E2 -14418.494} C_VEL
LIN {X 0,Y 485.778,Z 596.902,A -85,B 0,C 180,E1 -14421.13,E2 -14421.13} C_VEL
LIN {X 0,Y 485.777,Z 596.908,A -85,B 0,C 180,E1 -14423.812,E2 -14423.812} C_VEL
LIN {X 0,Y 485.789,Z 596.902,A -85,B 0,C 180,E1 -14426.625,E2 -14426.625} C_VEL
LIN {X 0,Y 485.786,Z 596.902,A -85,B 0,C 180,E1 -14429.356,E2 -14429.356} C_VEL
LIN {X 0,Y 485.722,Z 596.914,A -85,B 0,C 180,E1 -14432.247,E2 -14432.247} C_VEL
LIN {X 0,Y 485.758,Z 596.905,A -85,B 0,C 180,E1 -14435.225,E2 -14435.225} C_VEL
LIN {X 0,Y 485.767,Z 596.906,A -85,B 0,C 180,E1 -14437.527,E2 -14437.527} C_VEL
LIN {X 0,Y 485.734,Z 596.91,A -85,B 0,C 180,E1 -14440.46,E2 -14440.46} C_VEL
LIN {X 0,Y 485.787,Z 596.902,A -85,B 0,C 180,E1 -14442.663,E2 -14442.663} C_VEL
LIN {X 0,Y 485.775,Z 596.908,A -85,B 0,C 180,E1 -14446.202,E2 -14446.202} C_VEL
LIN {X 0,Y 485.758,Z 596.906,A -85,B 0,C 180,E1 -14448.575,E2 -14448.575} C_VEL
LIN {X 0,Y 485.718,Z 596.914,A -85,B 0,C 180,E1 -14451.677,E2 -14451.677} C_VEL
LIN {X 0,Y 485.733,Z 596.908,A -85,B 0,C 180,E1 -14454.773,E2 -14454.773} C_VEL
LIN {X 0,Y 485.721,Z 596.915,A -85,B 0,C 180,E1 -14457.753,E2 -14457.753} C_VEL
LIN {X 0,Y 485.781,Z 596.903,A -85,B 0,C 180,E1 -14460.644,E2 -14460.644} C_VEL
LIN {X 0,Y 485.763,Z 596.906,A -85,B 0,C 180,E1 -14463.449,E2 -14463.449} C_VEL
LIN {X 0,Y 485.819,Z 597.053,A -85,B 0,C 180,E1 -14465.017,E2 -14465.017} C_VEL
LIN {X 0,Y 488.164,Z 610.265,A -85,B 0,C 180,E1 -14467.652,E2 -14467.652} C_VEL
LIN {X 0,Y 487.839,Z 617.219,A -85,B 0,C 180,E1 -14468.964,E2 -14468.964} C_VEL
LIN {X 0,Y 486.659,Z 633.889,A -85,B 0,C 180,E1 -14472.071,E2 -14472.071} C_VEL
LIN {X 0,Y 486.009,Z 645.929,A -85,B 0,C 180,E1 -14474.301,E2 -14474.301} C_VEL
LIN {X 0,Y 489.178,Z 675.07,A -85,B 0,C 180,E1 -14474.916,E2 -14474.916} C_VEL
LIN {X 0,Y 487.896,Z 752.179,A -85,B 0,C 180,E1 -14476.298,E2 -14476.298} C_VEL
LIN {X 0,Y 487.69,Z 762.839,A -85,B 0,C 180,E1 -14476.583,E2 -14476.583} C_VEL
LIN {X 0,Y 487.308,Z 773.253,A -85,B 0,C 180,E1 -14476.969,E2 -14476.969} C_VEL
LIN {X 0,Y 486.96,Z 782.975,A -85,B 0,C 180,E1 -14477.434,E2 -14477.434} C_VEL
LIN {X 0,Y 486.57,Z 793.317,A -85,B 0,C 180,E1 -14478.058,E2 -14478.058} C_VEL
LIN {X 0,Y 486.114,Z 801.986,A -85,B 0,C 180,E1 -14478.689,E2 -14478.689} C_VEL
LIN {X 0,Y 485.64,Z 811.308,A -85,B 0,C 180,E1 -14479.509,E2 -14479.509} C_VEL
LIN {X 0,Y 485.193,Z 820.117,A -85,B 0,C 180,E1 -14480.444,E2 -14480.444} C_VEL
LIN {X 0,Y 484.818,Z 826.776,A -85,B 0,C 180,E1 -14481.275,E2 -14481.275} C_VEL
LIN {X 0,Y 484.52,Z 833.769,A -85,B 0,C 180,E1 -14482.315,E2 -14482.315} C_VEL
LIN {X 0,Y 484.288,Z 839.601,A -85,B 0,C 180,E1 -14483.356,E2 -14483.356} C_VEL
LIN {X 0,Y 484.123,Z 845.234,A -85,B 0,C 180,E1 -14484.604,E2 -14484.604} C_VEL
LIN {X 0,Y 484.042,Z 849.632,A -85,B 0,C 180,E1 -14485.851,E2 -14485.851} C_VEL
LIN {X 0,Y 483.968,Z 852.723,A -85,B 0,C 180,E1 -14487.003,E2 -14487.003} C_VEL
LIN {X 0,Y 483.968,Z 855.157,A -85,B 0,C 180,E1 -14488.341,E2 -14488.341} C_VEL
LIN {X 0,Y 484.006,Z 856.14,A -85,B 0,C 180,E1 -14489.171,E2 -14489.171} C_VEL
LIN {X 0,Y 483.967,Z 856.72,A -85,B 0,C 180,E1 -14490.829,E2 -14490.829} C_VEL
LIN {X 0,Y 483.935,Z 856.352,A -85,B 0,C 180,E1 -14491.659,E2 -14491.659} C_VEL
LIN {X 0,Y 483.976,Z 854.44,A -85,B 0,C 180,E1 -14493.319,E2 -14493.319} C_VEL
LIN {X 0,Y 484.029,Z 851.827,A -85,B 0,C 180,E1 -14494.565,E2 -14494.565} C_VEL
LIN {X 0,Y 484.256,Z 848.166,A -85,B 0,C 180,E1 -14495.811,E2 -14495.811} C_VEL
LIN {X 0,Y 484.506,Z 843.367,A -85,B 0,C 180,E1 -14497.059,E2 -14497.059} C_VEL
LIN {X 0,Y 484.97,Z 837.27,A -85,B 0,C 180,E1 -14498.304,E2 -14498.304} C_VEL
LIN {X 0,Y 485.52,Z 829.662,A -85,B 0,C 180,E1 -14499.55,E2 -14499.55} C_VEL
LIN {X 0,Y 486.189,Z 821.962,A -85,B 0,C 180,E1 -14500.585,E2 -14500.585} C_VEL
LIN {X 0,Y 486.879,Z 813.668,A -85,B 0,C 180,E1 -14501.514,E2 -14501.514} C_VEL
LIN {X 0,Y 487.52,Z 805.666,A -85,B 0,C 180,E1 -14502.273,E2 -14502.273} C_VEL
LIN {X 0,Y 488.224,Z 795.74,A -85,B 0,C 180,E1 -14503.06,E2 -14503.06} C_VEL
LIN {X 0,Y 488.866,Z 786.352,A -85,B 0,C 180,E1 -14503.675,E2 -14503.675} C_VEL
LIN {X 0,Y 489.496,Z 775.687,A -85,B 0,C 180,E1 -14504.238,E2 -14504.238} C_VEL
LIN {X 0,Y 490.178,Z 765.101,A -85,B 0,C 180,E1 -14504.667,E2 -14504.667} C_VEL
LIN {X 0,Y 490.68,Z 754.161,A -85,B 0,C 180,E1 -14504.995,E2 -14504.995} C_VEL
LIN {X 0,Y 491.15,Z 735.22,A -85,B 0,C 180,E1 -14505.377,E2 -14505.377} C_VEL
LIN {X 0,Y 492.549,Z 674.216,A -85,B 0,C 180,E1 -14506.54,E2 -14506.54} C_VEL
LIN {X 0,Y 490.175,Z 657.906,A -85,B 0,C 180,E1 -14506.999,E2 -14506.999} C_VEL
LIN {X 0,Y 487.465,Z 644.425,A -85,B 0,C 180,E1 -14507.444,E2 -14507.444} C_VEL
LIN {X 0,Y 488.896,Z 628.705,A -85,B 0,C 180,E1 -14510.55,E2 -14510.55} C_VEL
LIN {X 0,Y 489.988,Z 618.148,A -85,B 0,C 180,E1 -14512.704,E2 -14512.704} C_VEL
LIN {X 0,Y 488.377,Z 608.521,A -85,B 0,C 180,E1 -14514.928,E2 -14514.928} C_VEL
LIN {X 0,Y 486.511,Z 599.948,A -85,B 0,C 180,E1 -14517.056,E2 -14517.056} C_VEL
LIN {X 0,Y 485.774,Z 596.915,A -85,B 0,C 180,E1 -14517.887,E2 -14517.887} C_VEL
LIN {X 0,Y 485.77,Z 596.91,A -85,B 0,C 180,E1 -14520.31,E2 -14520.31} C_VEL
LIN {X 0,Y 485.757,Z 596.912,A -85,B 0,C 180,E1 -14523.245,E2 -14523.245} C_VEL
LIN {X 0,Y 485.809,Z 596.9,A -85,B 0,C 180,E1 -14526.238,E2 -14526.238} C_VEL
LIN {X 0,Y 485.766,Z 596.904,A -85,B 0,C 180,E1 -14529.38,E2 -14529.38} C_VEL
LIN {X 0,Y 485.789,Z 596.902,A -85,B 0,C 180,E1 -14532.663,E2 -14532.663} C_VEL
LIN {X 0,Y 485.792,Z 596.904,A -85,B 0,C 180,E1 -14535.048,E2 -14535.048} C_VEL
LIN {X 0,Y 485.788,Z 596.906,A -85,B 0,C 180,E1 -14538.451,E2 -14538.451} C_VEL
LIN {X 0,Y 485.774,Z 596.908,A -85,B 0,C 180,E1 -14541.136,E2 -14541.136} C_VEL
LIN {X 0,Y 485.817,Z 596.901,A -85,B 0,C 180,E1 -14543.843,E2 -14543.843} C_VEL
LIN {X 0,Y 485.796,Z 596.905,A -85,B 0,C 180,E1 -14546.777,E2 -14546.777} C_VEL
LIN {X 0,Y 485.793,Z 596.902,A -85,B 0,C 180,E1 -14549.896,E2 -14549.896} C_VEL
LIN {X 0,Y 485.822,Z 596.904,A -85,B 0,C 180,E1 -14552.525,E2 -14552.525} C_VEL
LIN {X 0,Y 485.79,Z 596.906,A -85,B 0,C 180,E1 -14555.283,E2 -14555.283} C_VEL
LIN {X 0,Y 485.806,Z 596.908,A -85,B 0,C 180,E1 -14557.983,E2 -14557.983} C_VEL
LIN {X 0,Y 485.832,Z 596.908,A -85,B 0,C 180,E1 -14560.634,E2 -14560.634} C_VEL
LIN {X 0,Y 485.809,Z 596.907,A -85,B 0,C 180,E1 -14563.24,E2 -14563.24} C_VEL
LIN {X 0,Y 485.905,Z 596.998,A -85,B 0,C 180,E1 -14565.158,E2 -14565.158} C_VEL
LIN {X 0,Y 487.924,Z 606.502,A -85,B 0,C 180,E1 -14567.806,E2 -14567.806} C_VEL
LIN {X 0,Y 489.132,Z 613.738,A -85,B 0,C 180,E1 -14569.688,E2 -14569.688} C_VEL
LIN {X 0,Y 488.903,Z 618.969,A -85,B 0,C 180,E1 -14570.932,E2 -14570.932} C_VEL
LIN {X 0,Y 488.091,Z 626.517,A -85,B 0,C 180,E1 -14572.657,E2 -14572.657} C_VEL
LIN {X 0,Y 491.929,Z 643.389,A -85,B 0,C 180,E1 -14573.228,E2 -14573.228} C_VEL
LIN {X 0,Y 493.106,Z 651.13,A -85,B 0,C 180,E1 -14573.449,E2 -14573.449} C_VEL
LIN {X 0,Y 491.18,Z 715.351,A -85,B 0,C 180,E1 -14574.656,E2 -14574.656} C_VEL
LIN {X 0,Y 490.66,Z 736.091,A -85,B 0,C 180,E1 -14575.086,E2 -14575.086} C_VEL
LIN {X 0,Y 490.014,Z 750.841,A -85,B 0,C 180,E1 -14575.593,E2 -14575.593} C_VEL
LIN {X 0,Y 489.539,Z 761.43,A -85,B 0,C 180,E1 -14576.103,E2 -14576.103} C_VEL
LIN {X 0,Y 489.008,Z 771.54,A -85,B 0,C 180,E1 -14576.715,E2 -14576.715} C_VEL
LIN {X 0,Y 488.404,Z 781.181,A -85,B 0,C 180,E1 -14577.431,E2 -14577.431} C_VEL
LIN {X 0,Y 487.66,Z 790.349,A -85,B 0,C 180,E1 -14578.251,E2 -14578.251} C_VEL
LIN {X 0,Y 486.928,Z 798.974,A -85,B 0,C 180,E1 -14579.176,E2 -14579.176} C_VEL
LIN {X 0,Y 486.271,Z 805.535,A -85,B 0,C 180,E1 -14580,E2 -14580} C_VEL
LIN {X 0,Y 485.667,Z 812.415,A -85,B 0,C 180,E1 -14581.033,E2 -14581.033} C_VEL
LIN {X 0,Y 485.174,Z 818.171,A -85,B 0,C 180,E1 -14582.068,E2 -14582.068} C_VEL
LIN {X 0,Y 484.704,Z 823.742,A -85,B 0,C 180,E1 -14583.313,E2 -14583.313} C_VEL
LIN {X 0,Y 484.49,Z 828.097,A -85,B 0,C 180,E1 -14584.56,E2 -14584.56} C_VEL
LIN {X 0,Y 484.233,Z 831.381,A -85,B 0,C 180,E1 -14585.811,E2 -14585.811} C_VEL
LIN {X 0,Y 484.085,Z 833.034,A -85,B 0,C 180,E1 -14586.647,E2 -14586.647} C_VEL
LIN {X 0,Y 483.883,Z 834.932,A -85,B 0,C 180,E1 -14588.323,E2 -14588.323} C_VEL
LIN {X 0,Y 483.869,Z 835.236,A -85,B 0,C 180,E1 -14589.162,E2 -14589.162} C_VEL
LIN {X 0,Y 483.868,Z 834.589,A -85,B 0,C 180,E1 -14590.847,E2 -14590.847} C_VEL
LIN {X 0,Y 483.847,Z 833.537,A -85,B 0,C 180,E1 -14591.693,E2 -14591.693} C_VEL
LIN {X 0,Y 483.974,Z 830.211,A -85,B 0,C 180,E1 -14593.389,E2 -14593.389} C_VEL
LIN {X 0,Y 484.154,Z 826.371,A -85,B 0,C 180,E1 -14594.665,E2 -14594.665} C_VEL
LIN {X 0,Y 484.332,Z 821.267,A -85,B 0,C 180,E1 -14595.948,E2 -14595.948} C_VEL
LIN {X 0,Y 484.622,Z 815.251,A -85,B 0,C 180,E1 -14597.147,E2 -14597.147} C_VEL
LIN {X 0,Y 484.831,Z 809.547,A -85,B 0,C 180,E1 -14598.096,E2 -14598.096} C_VEL
LIN {X 0,Y 485.241,Z 801.719,A -85,B 0,C 180,E1 -14599.171,E2 -14599.171} C_VEL
LIN {X 0,Y 485.663,Z 793.205,A -85,B 0,C 180,E1 -14600.141,E2 -14600.141} C_VEL
LIN {X 0,Y 486.042,Z 783.986,A -85,B 0,C 180,E1 -14601.013,E2 -14601.013} C_VEL
LIN {X 0,Y 486.522,Z 774.434,A -85,B 0,C 180,E1 -14601.76,E2 -14601.76} C_VEL
LIN {X 0,Y 486.937,Z 766.297,A -85,B 0,C 180,E1 -14602.296,E2 -14602.296} C_VEL
LIN {X 0,Y 487.328,Z 755.28,A -85,B 0,C 180,E1 -14602.88,E2 -14602.88} C_VEL
LIN {X 0,Y 487.569,Z 744.146,A -85,B 0,C 180,E1 -14603.336,E2 -14603.336} C_VEL
LIN {X 0,Y 487.859,Z 733.375,A -85,B 0,C 180,E1 -14603.656,E2 -14603.656} C_VEL
LIN {X 0,Y 488.299,Z 712.752,A -85,B 0,C 180,E1 -14604.046,E2 -14604.046} C_VEL
LIN {X 0,Y 489.308,Z 646.849,A -85,B 0,C 180,E1 -14605.221,E2 -14605.221} C_VEL
LIN {X 0,Y 486.217,Z 624.61,A -85,B 0,C 180,E1 -14605.72,E2 -14605.72} C_VEL
LIN {X 0,Y 486.949,Z 612.095,A -85,B 0,C 180,E1 -14608.338,E2 -14608.338} C_VEL
LIN {X 0,Y 487.245,Z 605.517,A -85,B 0,C 180,E1 -14609.732,E2 -14609.732} C_VEL
LIN {X 0,Y 485.846,Z 596.903,A -85,B 0,C 180,E1 -14611.646,E2 -14611.646} C_VEL
LIN {X 0,Y 485.787,Z 596.902,A -85,B 0,C 180,E1 -14614.727,E2 -14614.727} C_VEL
LIN {X 0,Y 485.774,Z 596.905,A -85,B 0,C 180,E1 -14617.528,E2 -14617.528} C_VEL
LIN {X 0,Y 485.791,Z 596.903,A -85,B 0,C 180,E1 -14620.453,E2 -14620.453} C_VEL
LIN {X 0,Y 485.786,Z 596.908,A -85,B 0,C 180,E1 -14623.868,E2 -14623.868} C_VEL
LIN {X 0,Y 485.787,Z 596.906,A -85,B 0,C 180,E1 -14626.203,E2 -14626.203} C_VEL
LIN {X 0,Y 485.79,Z 596.903,A -85,B 0,C 180,E1 -14629.546,E2 -14629.546} C_VEL
LIN {X 0,Y 485.795,Z 596.901,A -85,B 0,C 180,E1 -14632.729,E2 -14632.729} C_VEL
LIN {X 0,Y 485.798,Z 596.905,A -85,B 0,C 180,E1 -14635.783,E2 -14635.783} C_VEL
LIN {X 0,Y 485.78,Z 596.902,A -85,B 0,C 180,E1 -14638.729,E2 -14638.729} C_VEL
LIN {X 0,Y 485.801,Z 596.902,A -85,B 0,C 180,E1 -14641.588,E2 -14641.588} C_VEL
LIN {X 0,Y 485.769,Z 596.907,A -85,B 0,C 180,E1 -14644.368,E2 -14644.368} C_VEL
LIN {X 0,Y 485.784,Z 596.902,A -85,B 0,C 180,E1 -14647.338,E2 -14647.338} C_VEL
LIN {X 0,Y 485.841,Z 596.9,A -85,B 0,C 180,E1 -14649.756,E2 -14649.756} C_VEL
LIN {X 0,Y 485.857,Z 596.896,A -85,B 0,C 180,E1 -14652.377,E2 -14652.377} C_VEL
LIN {X 0,Y 485.934,Z 596.883,A -85,B 0,C 180,E1 -14654.962,E2 -14654.962} C_VEL
LIN {X 0,Y 485.934,Z 596.884,A -85,B 0,C 180,E1 -14658.57,E2 -14658.57} C_VEL
LIN {X 0,Y 485.934,Z 596.887,A -85,B 0,C 180,E1 -14661.712,E2 -14661.712} C_VEL
LIN {X 0,Y 486.072,Z 596.866,A -85,B 0,C 180,E1 -14665.04,E2 -14665.04} C_VEL
LIN {X 0,Y 485.903,Z 596.89,A -85,B 0,C 180,E1 -14668.348,E2 -14668.348} C_VEL
LIN {X 0,Y 486.134,Z 596.866,A -85,B 0,C 180,E1 -14670,E2 -14670} C_VEL
LIN {X 0,Y 486.034,Z 596.877,A -85,B 0,C 180,E1 -14674.132,E2 -14674.132} C_VEL
LIN {X 0,Y 485.986,Z 596.877,A -85,B 0,C 180,E1 -14676.621,E2 -14676.621} C_VEL
LIN {X 0,Y 485.913,Z 596.885,A -85,B 0,C 180,E1 -14679.123,E2 -14679.123} C_VEL
LIN {X 0,Y 485.911,Z 596.889,A -85,B 0,C 180,E1 -14681.643,E2 -14681.643} C_VEL
LIN {X 0,Y 485.934,Z 596.883,A -85,B 0,C 180,E1 -14685.038,E2 -14685.038} C_VEL
LIN {X 0,Y 485.825,Z 596.897,A -85,B 0,C 180,E1 -14687.248,E2 -14687.248} C_VEL
LIN {X 0,Y 485.192,Z 596.983,A -85,B 0,C 180,E1 -14687.94,E2 -14687.94} C_VEL
LIN {X 0,Y 482.347,Z 597.333,A -85,B 0,C 180,E1 -14689.064,E2 -14689.064} C_VEL
LIN {X 0,Y 479.914,Z 597.641,A -85,B 0,C 180,E1 -14689.97,E2 -14689.97} C_VEL
LIN {X 0,Y 478.859,Z 597.765,A -85,B 0,C 180,E1 -14690.67,E2 -14690.67} C_VEL
LIN {X 0,Y 478.769,Z 597.775,A -85,B 0,C 180,E1 -14690.907,E2 -14690.907} C_VEL
LIN {X 0,Y 478.738,Z 597.78,A -85,B 0,C 180,E1 -14693.268,E2 -14693.268} C_VEL
LIN {X 0,Y 478.741,Z 597.787,A -85,B 0,C 180,E1 -14696.035,E2 -14696.035} C_VEL
LIN {X 0,Y 478.75,Z 597.778,A -85,B 0,C 180,E1 -14698.869,E2 -14698.869} C_VEL
LIN {X 0,Y 478.756,Z 597.785,A -85,B 0,C 180,E1 -14701.945,E2 -14701.945} C_VEL
LIN {X 0,Y 478.767,Z 597.776,A -85,B 0,C 180,E1 -14704.987,E2 -14704.987} C_VEL
LIN {X 0,Y 478.757,Z 597.784,A -85,B 0,C 180,E1 -14707.914,E2 -14707.914} C_VEL
LIN {X 0,Y 478.74,Z 597.779,A -85,B 0,C 180,E1 -14711.177,E2 -14711.177} C_VEL
LIN {X 0,Y 478.747,Z 597.779,A -85,B 0,C 180,E1 -14714.61,E2 -14714.61} C_VEL
LIN {X 0,Y 478.725,Z 597.785,A -85,B 0,C 180,E1 -14717.698,E2 -14717.698} C_VEL
LIN {X 0,Y 478.764,Z 597.776,A -85,B 0,C 180,E1 -14720.842,E2 -14720.842} C_VEL
LIN {X 0,Y 478.798,Z 597.775,A -85,B 0,C 180,E1 -14723.572,E2 -14723.572} C_VEL
LIN {X 0,Y 478.751,Z 597.779,A -85,B 0,C 180,E1 -14726.506,E2 -14726.506} C_VEL
LIN {X 0,Y 478.734,Z 597.784,A -85,B 0,C 180,E1 -14729.682,E2 -14729.682} C_VEL
LIN {X 0,Y 478.761,Z 597.783,A -85,B 0,C 180,E1 -14732.085,E2 -14732.085} C_VEL
LIN {X 0,Y 478.745,Z 597.778,A -85,B 0,C 180,E1 -14735.109,E2 -14735.109} C_VEL
LIN {X 0,Y 478.773,Z 597.776,A -85,B 0,C 180,E1 -14738.547,E2 -14738.547} C_VEL
LIN {X 0,Y 478.784,Z 597.774,A -85,B 0,C 180,E1 -14741.225,E2 -14741.225} C_VEL
LIN {X 0,Y 478.83,Z 597.768,A -85,B 0,C 180,E1 -14744.898,E2 -14744.898} C_VEL
LIN {X 0,Y 478.871,Z 597.768,A -85,B 0,C 180,E1 -14748.184,E2 -14748.184} C_VEL
LIN {X 0,Y 478.911,Z 597.761,A -85,B 0,C 180,E1 -14751.59,E2 -14751.59} C_VEL
LIN {X 0,Y 479.008,Z 597.752,A -85,B 0,C 180,E1 -14754.125,E2 -14754.125} C_VEL
LIN {X 0,Y 478.956,Z 597.753,A -85,B 0,C 180,E1 -14756.647,E2 -14756.647} C_VEL
LIN {X 0,Y 479.09,Z 597.744,A -85,B 0,C 180,E1 -14760,E2 -14760} C_VEL
LIN {X 0,Y 478.992,Z 597.753,A -85,B 0,C 180,E1 -14764.193,E2 -14764.193} C_VEL
LIN {X 0,Y 478.941,Z 597.755,A -85,B 0,C 180,E1 -14766.719,E2 -14766.719} C_VEL
LIN {X 0,Y 478.871,Z 597.763,A -85,B 0,C 180,E1 -14769.259,E2 -14769.259} C_VEL
LIN {X 0,Y 478.869,Z 597.769,A -85,B 0,C 180,E1 -14771.817,E2 -14771.817} C_VEL
LIN {X 0,Y 478.822,Z 597.769,A -85,B 0,C 180,E1 -14775.098,E2 -14775.098} C_VEL
LIN {X 0,Y 478.775,Z 597.783,A -85,B 0,C 180,E1 -14778.021,E2 -14778.021} C_VEL
LIN {X 0,Y 478.75,Z 597.779,A -85,B 0,C 180,E1 -14780.557,E2 -14780.557} C_VEL
LIN {X 0,Y 478.74,Z 597.78,A -85,B 0,C 180,E1 -14783.268,E2 -14783.268} C_VEL
LIN {X 0,Y 478.731,Z 597.788,A -85,B 0,C 180,E1 -14786.036,E2 -14786.036} C_VEL
LIN {X 0,Y 478.742,Z 597.779,A -85,B 0,C 180,E1 -14788.87,E2 -14788.87} C_VEL
LIN {X 0,Y 478.674,Z 597.795,A -85,B 0,C 180,E1 -14791.928,E2 -14791.928} C_VEL
LIN {X 0,Y 478.722,Z 597.781,A -85,B 0,C 180,E1 -14794.979,E2 -14794.979} C_VEL
LIN {X 0,Y 478.695,Z 597.792,A -85,B 0,C 180,E1 -14797.92,E2 -14797.92} C_VEL
LIN {X 0,Y 478.71,Z 597.783,A -85,B 0,C 180,E1 -14801.181,E2 -14801.181} C_VEL
LIN {X 0,Y 478.731,Z 597.785,A -85,B 0,C 180,E1 -14804.198,E2 -14804.198} C_VEL
LIN {X 0,Y 478.72,Z 597.781,A -85,B 0,C 180,E1 -14807.019,E2 -14807.019} C_VEL
LIN {X 0,Y 478.689,Z 597.793,A -85,B 0,C 180,E1 -14809.922,E2 -14809.922} C_VEL
LIN {X 0,Y 478.671,Z 597.788,A -85,B 0,C 180,E1 -14813.133,E2 -14813.133} C_VEL
LIN {X 0,Y 478.694,Z 597.79,A -85,B 0,C 180,E1 -14816.218,E2 -14816.218} C_VEL
LIN {X 0,Y 478.715,Z 597.786,A -85,B 0,C 180,E1 -14819.686,E2 -14819.686} C_VEL
LIN {X 0,Y 478.736,Z 597.786,A -85,B 0,C 180,E1 -14822.083,E2 -14822.083} C_VEL
LIN {X 0,Y 478.746,Z 597.898,A -85,B 0,C 180,E1 -14824.894,E2 -14824.894} C_VEL
LIN {X 0,Y 481.099,Z 610.906,A -85,B 0,C 180,E1 -14827.531,E2 -14827.531} C_VEL
LIN {X 0,Y 481.017,Z 615.546,A -85,B 0,C 180,E1 -14828.427,E2 -14828.427} C_VEL
LIN {X 0,Y 479.94,Z 630.552,A -85,B 0,C 180,E1 -14831.272,E2 -14831.272} C_VEL
LIN {X 0,Y 478.989,Z 645.804,A -85,B 0,C 180,E1 -14834.139,E2 -14834.139} C_VEL
LIN {X 0,Y 482.175,Z 675.613,A -85,B 0,C 180,E1 -14834.778,E2 -14834.778} C_VEL
LIN {X 0,Y 480.88,Z 752.015,A -85,B 0,C 180,E1 -14836.174,E2 -14836.174} C_VEL
LIN {X 0,Y 480.679,Z 762.662,A -85,B 0,C 180,E1 -14836.464,E2 -14836.464} C_VEL
LIN {X 0,Y 480.312,Z 772.487,A -85,B 0,C 180,E1 -14836.829,E2 -14836.829} C_VEL
LIN {X 0,Y 480.018,Z 781.417,A -85,B 0,C 180,E1 -14837.25,E2 -14837.25} C_VEL
LIN {X 0,Y 479.555,Z 792.005,A -85,B 0,C 180,E1 -14837.88,E2 -14837.88} C_VEL
LIN {X 0,Y 479.037,Z 802.11,A -85,B 0,C 180,E1 -14838.625,E2 -14838.625} C_VEL
LIN {X 0,Y 478.57,Z 811.404,A -85,B 0,C 180,E1 -14839.458,E2 -14839.458} C_VEL
LIN {X 0,Y 478.181,Z 819.312,A -85,B 0,C 180,E1 -14840.302,E2 -14840.302} C_VEL
LIN {X 0,Y 477.784,Z 826.078,A -85,B 0,C 180,E1 -14841.145,E2 -14841.145} C_VEL
LIN {X 0,Y 477.458,Z 833.167,A -85,B 0,C 180,E1 -14842.201,E2 -14842.201} C_VEL
LIN {X 0,Y 477.231,Z 839.086,A -85,B 0,C 180,E1 -14843.257,E2 -14843.257} C_VEL
LIN {X 0,Y 477.061,Z 844.798,A -85,B 0,C 180,E1 -14844.524,E2 -14844.524} C_VEL
LIN {X 0,Y 476.955,Z 849.26,A -85,B 0,C 180,E1 -14845.789,E2 -14845.789} C_VEL
LIN {X 0,Y 476.892,Z 852.787,A -85,B 0,C 180,E1 -14847.149,E2 -14847.149} C_VEL
LIN {X 0,Y 476.877,Z 854.902,A -85,B 0,C 180,E1 -14848.317,E2 -14848.317} C_VEL
LIN {X 0,Y 476.909,Z 855.882,A -85,B 0,C 180,E1 -14849.159,E2 -14849.159} C_VEL
LIN {X 0,Y 476.871,Z 856.582,A -85,B 0,C 180,E1 -14850.842,E2 -14850.842} C_VEL
LIN {X 0,Y 476.853,Z 855.467,A -85,B 0,C 180,E1 -14852.526,E2 -14852.526} C_VEL
LIN {X 0,Y 476.887,Z 854.398,A -85,B 0,C 180,E1 -14853.368,E2 -14853.368} C_VEL
LIN {X 0,Y 476.96,Z 851.832,A -85,B 0,C 180,E1 -14854.633,E2 -14854.633} C_VEL
LIN {X 0,Y 477.178,Z 848.225,A -85,B 0,C 180,E1 -14855.898,E2 -14855.898} C_VEL
LIN {X 0,Y 477.458,Z 843.491,A -85,B 0,C 180,E1 -14857.163,E2 -14857.163} C_VEL
LIN {X 0,Y 478.015,Z 836.272,A -85,B 0,C 180,E1 -14858.638,E2 -14858.638} C_VEL
LIN {X 0,Y 478.525,Z 829.932,A -85,B 0,C 180,E1 -14859.691,E2 -14859.691} C_VEL
LIN {X 0,Y 479.236,Z 822.338,A -85,B 0,C 180,E1 -14860.74,E2 -14860.74} C_VEL
LIN {X 0,Y 479.95,Z 814.199,A -85,B 0,C 180,E1 -14861.683,E2 -14861.683} C_VEL
LIN {X 0,Y 480.636,Z 806.172,A -85,B 0,C 180,E1 -14862.47,E2 -14862.47} C_VEL
LIN {X 0,Y 481.388,Z 796.664,A -85,B 0,C 180,E1 -14863.248,E2 -14863.248} C_VEL
LIN {X 0,Y 482.039,Z 787.526,A -85,B 0,C 180,E1 -14863.873,E2 -14863.873} C_VEL
LIN {X 0,Y 482.765,Z 776.068,A -85,B 0,C 180,E1 -14864.494,E2 -14864.494} C_VEL
LIN {X 0,Y 483.476,Z 764.924,A -85,B 0,C 180,E1 -14864.955,E2 -14864.955} C_VEL
LIN {X 0,Y 484.036,Z 754.004,A -85,B 0,C 180,E1 -14865.286,E2 -14865.286} C_VEL
LIN {X 0,Y 484.53,Z 735.189,A -85,B 0,C 180,E1 -14865.673,E2 -14865.673} C_VEL
LIN {X 0,Y 485.986,Z 674.967,A -85,B 0,C 180,E1 -14866.85,E2 -14866.85} C_VEL
LIN {X 0,Y 483.655,Z 658.968,A -85,B 0,C 180,E1 -14867.324,E2 -14867.324} C_VEL
LIN {X 0,Y 480.644,Z 644.269,A -85,B 0,C 180,E1 -14867.821,E2 -14867.821} C_VEL
LIN {X 0,Y 482.246,Z 628.194,A -85,B 0,C 180,E1 -14871.069,E2 -14871.069} C_VEL
LIN {X 0,Y 483.152,Z 619.76,A -85,B 0,C 180,E1 -14872.818,E2 -14872.818} C_VEL
LIN {X 0,Y 481.637,Z 610.768,A -85,B 0,C 180,E1 -14874.945,E2 -14874.945} C_VEL
LIN {X 0,Y 479.555,Z 601.161,A -85,B 0,C 180,E1 -14877.393,E2 -14877.393} C_VEL
LIN {X 0,Y 478.762,Z 597.788,A -85,B 0,C 180,E1 -14878.348,E2 -14878.348} C_VEL
LIN {X 0,Y 478.709,Z 597.79,A -85,B 0,C 180,E1 -14880.805,E2 -14880.805} C_VEL
LIN {X 0,Y 478.711,Z 597.789,A -85,B 0,C 180,E1 -14883.781,E2 -14883.781} C_VEL
LIN {X 0,Y 478.74,Z 597.78,A -85,B 0,C 180,E1 -14886.861,E2 -14886.861} C_VEL
LIN {X 0,Y 478.723,Z 597.778,A -85,B 0,C 180,E1 -14890.075,E2 -14890.075} C_VEL
LIN {X 0,Y 478.748,Z 597.779,A -85,B 0,C 180,E1 -14893.444,E2 -14893.444} C_VEL
LIN {X 0,Y 478.749,Z 597.783,A -85,B 0,C 180,E1 -14896.556,E2 -14896.556} C_VEL
LIN {X 0,Y 478.765,Z 597.78,A -85,B 0,C 180,E1 -14899.929,E2 -14899.929} C_VEL
LIN {X 0,Y 478.754,Z 597.782,A -85,B 0,C 180,E1 -14903.58,E2 -14903.58} C_VEL
LIN {X 0,Y 478.757,Z 597.78,A -85,B 0,C 180,E1 -14906.506,E2 -14906.506} C_VEL
LIN {X 0,Y 478.73,Z 597.785,A -85,B 0,C 180,E1 -14909.196,E2 -14909.196} C_VEL
LIN {X 0,Y 478.774,Z 597.779,A -85,B 0,C 180,E1 -14912.085,E2 -14912.085} C_VEL
LIN {X 0,Y 478.749,Z 597.785,A -85,B 0,C 180,E1 -14915.109,E2 -14915.109} C_VEL
LIN {X 0,Y 478.777,Z 597.785,A -85,B 0,C 180,E1 -14918.546,E2 -14918.546} C_VEL
LIN {X 0,Y 478.789,Z 597.785,A -85,B 0,C 180,E1 -14921.225,E2 -14921.225} C_VEL
LIN {X 0,Y 478.859,Z 597.91,A -85,B 0,C 180,E1 -14924.734,E2 -14924.734} C_VEL
LIN {X 0,Y 481.072,Z 608.091,A -85,B 0,C 180,E1 -14927.646,E2 -14927.646} C_VEL
LIN {X 0,Y 482.272,Z 615.214,A -85,B 0,C 180,E1 -14929.54,E2 -14929.54} C_VEL
LIN {X 0,Y 482.062,Z 620.415,A -85,B 0,C 180,E1 -14930.803,E2 -14930.803} C_VEL
LIN {X 0,Y 481.306,Z 626.777,A -85,B 0,C 180,E1 -14932.283,E2 -14932.283} C_VEL
LIN {X 0,Y 485.197,Z 643.152,A -85,B 0,C 180,E1 -14932.86,E2 -14932.86} C_VEL
LIN {X 0,Y 486.587,Z 651.956,A -85,B 0,C 180,E1 -14933.127,E2 -14933.127} C_VEL
LIN {X 0,Y 484.624,Z 713.62,A -85,B 0,C 180,E1 -14934.323,E2 -14934.323} C_VEL
LIN {X 0,Y 484.066,Z 734.719,A -85,B 0,C 180,E1 -14934.759,E2 -14934.759} C_VEL
LIN {X 0,Y 483.549,Z 747.669,A -85,B 0,C 180,E1 -14935.17,E2 -14935.17} C_VEL
LIN {X 0,Y 482.917,Z 760.078,A -85,B 0,C 180,E1 -14935.737,E2 -14935.737} C_VEL
LIN {X 0,Y 482.249,Z 771.931,A -85,B 0,C 180,E1 -14936.461,E2 -14936.461} C_VEL
LIN {X 0,Y 481.629,Z 781.536,A -85,B 0,C 180,E1 -14937.186,E2 -14937.186} C_VEL
LIN {X 0,Y 480.841,Z 790.688,A -85,B 0,C 180,E1 -14938.017,E2 -14938.017} C_VEL
LIN {X 0,Y 480.241,Z 797.56,A -85,B 0,C 180,E1 -14938.746,E2 -14938.746} C_VEL
LIN {X 0,Y 479.378,Z 805.784,A -85,B 0,C 180,E1 -14939.79,E2 -14939.79} C_VEL
LIN {X 0,Y 478.711,Z 812.633,A -85,B 0,C 180,E1 -14940.838,E2 -14940.838} C_VEL
LIN {X 0,Y 478.316,Z 817.35,A -85,B 0,C 180,E1 -14941.678,E2 -14941.678} C_VEL
LIN {X 0,Y 477.721,Z 823.174,A -85,B 0,C 180,E1 -14942.941,E2 -14942.941} C_VEL
LIN {X 0,Y 477.501,Z 827.713,A -85,B 0,C 180,E1 -14944.206,E2 -14944.206} C_VEL
LIN {X 0,Y 477.16,Z 831.442,A -85,B 0,C 180,E1 -14945.656,E2 -14945.656} C_VEL
LIN {X 0,Y 476.97,Z 833.587,A -85,B 0,C 180,E1 -14946.747,E2 -14946.747} C_VEL
LIN {X 0,Y 476.792,Z 835.187,A -85,B 0,C 180,E1 -14948.447,E2 -14948.447} C_VEL
LIN {X 0,Y 476.786,Z 835.469,A -85,B 0,C 180,E1 -14949.299,E2 -14949.299} C_VEL
LIN {X 0,Y 476.829,Z 835.115,A -85,B 0,C 180,E1 -14950.196,E2 -14950.196} C_VEL
LIN {X 0,Y 476.751,Z 833.413,A -85,B 0,C 180,E1 -14951.869,E2 -14951.869} C_VEL
LIN {X 0,Y 476.851,Z 830.864,A -85,B 0,C 180,E1 -14953.16,E2 -14953.16} C_VEL
LIN {X 0,Y 477.06,Z 827.224,A -85,B 0,C 180,E1 -14954.454,E2 -14954.454} C_VEL
LIN {X 0,Y 477.257,Z 821.345,A -85,B 0,C 180,E1 -14955.973,E2 -14955.973} C_VEL
LIN {X 0,Y 477.498,Z 816.049,A -85,B 0,C 180,E1 -14957.06,E2 -14957.06} C_VEL
LIN {X 0,Y 477.745,Z 809.582,A -85,B 0,C 180,E1 -14958.153,E2 -14958.153} C_VEL
LIN {X 0,Y 478.181,Z 801.734,A -85,B 0,C 180,E1 -14959.243,E2 -14959.243} C_VEL
LIN {X 0,Y 478.564,Z 794.272,A -85,B 0,C 180,E1 -14960.118,E2 -14960.118} C_VEL
LIN {X 0,Y 478.938,Z 785.313,A -85,B 0,C 180,E1 -14960.996,E2 -14960.996} C_VEL
LIN {X 0,Y 479.445,Z 775.928,A -85,B 0,C 180,E1 -14961.759,E2 -14961.759} C_VEL
LIN {X 0,Y 479.907,Z 766.158,A -85,B 0,C 180,E1 -14962.414,E2 -14962.414} C_VEL
LIN {X 0,Y 480.325,Z 754.859,A -85,B 0,C 180,E1 -14963.016,E2 -14963.016} C_VEL
LIN {X 0,Y 480.542,Z 744.338,A -85,B 0,C 180,E1 -14963.452,E2 -14963.452} C_VEL
LIN {X 0,Y 480.842,Z 734.021,A -85,B 0,C 180,E1 -14963.767,E2 -14963.767} C_VEL
LIN {X 0,Y 481.278,Z 713.811,A -85,B 0,C 180,E1 -14964.162,E2 -14964.162} C_VEL
LIN {X 0,Y 482.316,Z 647.575,A -85,B 0,C 180,E1 -14965.363,E2 -14965.363} C_VEL
LIN {X 0,Y 479.201,Z 624.789,A -85,B 0,C 180,E1 -14965.878,E2 -14965.878} C_VEL
LIN {X 0,Y 480.003,Z 611.084,A -85,B 0,C 180,E1 -14968.786,E2 -14968.786} C_VEL
LIN {X 0,Y 480.238,Z 606.7,A -85,B 0,C 180,E1 -14969.729,E2 -14969.729} C_VEL
LIN {X 0,Y 478.796,Z 597.781,A -85,B 0,C 180,E1 -14971.779,E2 -14971.779} C_VEL
LIN {X 0,Y 478.743,Z 597.778,A -85,B 0,C 180,E1 -14974.982,E2 -14974.982} C_VEL
LIN {X 0,Y 478.713,Z 597.79,A -85,B 0,C 180,E1 -14977.918,E2 -14977.918} C_VEL
LIN {X 0,Y 478.754,Z 597.779,A -85,B 0,C 180,E1 -14980.466,E2 -14980.466} C_VEL
LIN {X 0,Y 478.747,Z 597.78,A -85,B 0,C 180,E1 -14983.443,E2 -14983.443} C_VEL
LIN {X 0,Y 478.746,Z 597.78,A -85,B 0,C 180,E1 -14986.556,E2 -14986.556} C_VEL
LIN {X 0,Y 478.761,Z 597.784,A -85,B 0,C 180,E1 -14989.929,E2 -14989.929} C_VEL
LIN {X 0,Y 478.749,Z 597.781,A -85,B 0,C 180,E1 -14993.579,E2 -14993.579} C_VEL
LIN {X 0,Y 478.751,Z 597.779,A -85,B 0,C 180,E1 -14996.505,E2 -14996.505} C_VEL
LIN {X 0,Y 478.731,Z 597.784,A -85,B 0,C 180,E1 -14999.682,E2 -14999.682} C_VEL
LIN {X 0,Y 478.759,Z 597.784,A -85,B 0,C 180,E1 -15002.084,E2 -15002.084} C_VEL
LIN {X 0,Y 478.743,Z 597.779,A -85,B 0,C 180,E1 -15005.108,E2 -15005.108} C_VEL
LIN {X 0,Y 478.771,Z 597.777,A -85,B 0,C 180,E1 -15008.546,E2 -15008.546} C_VEL
LIN {X 0,Y 478.815,Z 597.778,A -85,B 0,C 180,E1 -15011.963,E2 -15011.963} C_VEL
LIN {X 0,Y 478.861,Z 597.767,A -85,B 0,C 180,E1 -15015.601,E2 -15015.601} C_VEL
LIN {X 0,Y 478.907,Z 597.758,A -85,B 0,C 180,E1 -15019.039,E2 -15019.039} C_VEL
LIN {X 0,Y 478.926,Z 597.758,A -85,B 0,C 180,E1 -15022.436,E2 -15022.436} C_VEL
LIN {X 0,Y 479.03,Z 597.743,A -85,B 0,C 180,E1 -15024.967,E2 -15024.967} C_VEL
LIN {X 0,Y 478.818,Z 597.771,A -85,B 0,C 180,E1 -15027.485,E2 -15027.485} C_VEL
LIN {X 0,Y 479.088,Z 597.744,A -85,B 0,C 180,E1 -15030,E2 -15030} C_VEL
LIN {X 0,Y 479,Z 597.752,A -85,B 0,C 180,E1 -15034.193,E2 -15034.193} C_VEL
LIN {X 0,Y 478.936,Z 597.755,A -85,B 0,C 180,E1 -15036.719,E2 -15036.719} C_VEL
LIN {X 0,Y 478.865,Z 597.764,A -85,B 0,C 180,E1 -15039.259,E2 -15039.259} C_VEL
LIN {X 0,Y 478.869,Z 597.769,A -85,B 0,C 180,E1 -15041.816,E2 -15041.816} C_VEL
LIN {X 0,Y 478.874,Z 597.763,A -85,B 0,C 180,E1 -15045.265,E2 -15045.265} C_VEL
LIN {X 0,Y 478.784,Z 597.774,A -85,B 0,C 180,E1 -15048.775,E2 -15048.775} C_VEL
LIN {X 0,Y 478.769,Z 597.775,A -85,B 0,C 180,E1 -15050.907,E2 -15050.907} C_VEL
LIN {X 0,Y 478.088,Z 597.865,A -85,B 0,C 180,E1 -15051.609,E2 -15051.609} C_VEL
LIN {X 0,Y 475.219,Z 598.221,A -85,B 0,C 180,E1 -15052.749,E2 -15052.749} C_VEL
LIN {X 0,Y 472.802,Z 598.523,A -85,B 0,C 180,E1 -15053.668,E2 -15053.668} C_VEL
LIN {X 0,Y 471.767,Z 598.651,A -85,B 0,C 180,E1 -15054.378,E2 -15054.378} C_VEL
LIN {X 0,Y 471.684,Z 598.659,A -85,B 0,C 180,E1 -15054.618,E2 -15054.618} C_VEL
LIN {X 0,Y 471.71,Z 598.656,A -85,B 0,C 180,E1 -15057.408,E2 -15057.408} C_VEL
LIN {X 0,Y 471.718,Z 598.655,A -85,B 0,C 180,E1 -15060.546,E2 -15060.546} C_VEL
LIN {X 0,Y 471.741,Z 598.656,A -85,B 0,C 180,E1 -15063.749,E2 -15063.749} C_VEL
LIN {X 0,Y 471.75,Z 598.651,A -85,B 0,C 180,E1 -15066.7,E2 -15066.7} C_VEL
LIN {X 0,Y 471.724,Z 598.657,A -85,B 0,C 180,E1 -15069.679,E2 -15069.679} C_VEL
LIN {X 0,Y 471.689,Z 598.658,A -85,B 0,C 180,E1 -15073.312,E2 -15073.312} C_VEL
LIN {X 0,Y 471.698,Z 598.661,A -85,B 0,C 180,E1 -15075.74,E2 -15075.74} C_VEL
LIN {X 0,Y 471.702,Z 598.656,A -85,B 0,C 180,E1 -15079.228,E2 -15079.228} C_VEL
LIN {X 0,Y 471.7,Z 598.663,A -85,B 0,C 180,E1 -15081.907,E2 -15081.907} C_VEL
LIN {X 0,Y 471.694,Z 598.657,A -85,B 0,C 180,E1 -15084.758,E2 -15084.758} C_VEL
LIN {X 0,Y 471.688,Z 598.664,A -85,B 0,C 180,E1 -15087.826,E2 -15087.826} C_VEL
LIN {X 0,Y 471.689,Z 598.658,A -85,B 0,C 180,E1 -15090.657,E2 -15090.657} C_VEL
LIN {X 0,Y 471.699,Z 598.659,A -85,B 0,C 180,E1 -15093.546,E2 -15093.546} C_VEL
LIN {X 0,Y 471.676,Z 598.662,A -85,B 0,C 180,E1 -15096.363,E2 -15096.363} C_VEL
LIN {X 0,Y 471.754,Z 598.65,A -85,B 0,C 180,E1 -15099.293,E2 -15099.293} C_VEL
LIN {X 0,Y 471.758,Z 598.655,A -85,B 0,C 180,E1 -15101.849,E2 -15101.849} C_VEL
LIN {X 0,Y 471.783,Z 598.647,A -85,B 0,C 180,E1 -15105.381,E2 -15105.381} C_VEL
LIN {X 0,Y 471.854,Z 598.637,A -85,B 0,C 180,E1 -15108.874,E2 -15108.874} C_VEL
LIN {X 0,Y 471.889,Z 598.636,A -85,B 0,C 180,E1 -15112.323,E2 -15112.323} C_VEL
LIN {X 0,Y 471.972,Z 598.622,A -85,B 0,C 180,E1 -15114.892,E2 -15114.892} C_VEL
LIN {X 0,Y 471.795,Z 598.646,A -85,B 0,C 180,E1 -15117.448,E2 -15117.448} C_VEL
LIN {X 0,Y 472.044,Z 598.621,A -85,B 0,C 180,E1 -15120,E2 -15120} C_VEL
LIN {X 0,Y 471.96,Z 598.628,A -85,B 0,C 180,E1 -15124.256,E2 -15124.256} C_VEL
LIN {X 0,Y 471.893,Z 598.632,A -85,B 0,C 180,E1 -15126.82,E2 -15126.82} C_VEL
LIN {X 0,Y 471.835,Z 598.64,A -85,B 0,C 180,E1 -15129.398,E2 -15129.398} C_VEL
LIN {X 0,Y 471.819,Z 598.649,A -85,B 0,C 180,E1 -15131.996,E2 -15131.996} C_VEL
LIN {X 0,Y 471.769,Z 598.648,A -85,B 0,C 180,E1 -15135.189,E2 -15135.189} C_VEL
LIN {X 0,Y 471.73,Z 598.658,A -85,B 0,C 180,E1 -15138.169,E2 -15138.169} C_VEL
LIN {X 0,Y 471.708,Z 598.655,A -85,B 0,C 180,E1 -15140.878,E2 -15140.878} C_VEL
LIN {X 0,Y 471.676,Z 598.663,A -85,B 0,C 180,E1 -15143.638,E2 -15143.638} C_VEL
LIN {X 0,Y 471.688,Z 598.66,A -85,B 0,C 180,E1 -15146.455,E2 -15146.455} C_VEL
LIN {X 0,Y 471.682,Z 598.659,A -85,B 0,C 180,E1 -15149.344,E2 -15149.344} C_VEL
LIN {X 0,Y 471.623,Z 598.669,A -85,B 0,C 180,E1 -15152.321,E2 -15152.321} C_VEL
LIN {X 0,Y 471.675,Z 598.66,A -85,B 0,C 180,E1 -15155.391,E2 -15155.391} C_VEL
LIN {X 0,Y 471.635,Z 598.665,A -85,B 0,C 180,E1 -15158.591,E2 -15158.591} C_VEL
LIN {X 0,Y 471.668,Z 598.668,A -85,B 0,C 180,E1 -15161.933,E2 -15161.933} C_VEL
LIN {X 0,Y 471.706,Z 598.657,A -85,B 0,C 180,E1 -15164.54,E2 -15164.54} C_VEL
LIN {X 0,Y 471.669,Z 598.668,A -85,B 0,C 180,E1 -15167.946,E2 -15167.946} C_VEL
LIN {X 0,Y 471.642,Z 598.665,A -85,B 0,C 180,E1 -15170.557,E2 -15170.557} C_VEL
LIN {X 0,Y 471.625,Z 598.668,A -85,B 0,C 180,E1 -15173.554,E2 -15173.554} C_VEL
LIN {X 0,Y 471.66,Z 598.665,A -85,B 0,C 180,E1 -15176.267,E2 -15176.267} C_VEL
LIN {X 0,Y 471.68,Z 598.662,A -85,B 0,C 180,E1 -15179.675,E2 -15179.675} C_VEL
LIN {X 0,Y 471.681,Z 598.66,A -85,B 0,C 180,E1 -15182.591,E2 -15182.591} C_VEL
LIN {X 0,Y 471.71,Z 598.798,A -85,B 0,C 180,E1 -15184.787,E2 -15184.787} C_VEL
LIN {X 0,Y 474.171,Z 612.708,A -85,B 0,C 180,E1 -15187.643,E2 -15187.643} C_VEL
LIN {X 0,Y 473.294,Z 625.413,A -85,B 0,C 180,E1 -15190.1,E2 -15190.1} C_VEL
LIN {X 0,Y 472.041,Z 643.84,A -85,B 0,C 180,E1 -15193.624,E2 -15193.624} C_VEL
LIN {X 0,Y 471.944,Z 645.709,A -85,B 0,C 180,E1 -15193.978,E2 -15193.978} C_VEL
LIN {X 0,Y 475.208,Z 675.002,A -85,B 0,C 180,E1 -15194.614,E2 -15194.614} C_VEL
LIN {X 0,Y 473.833,Z 752.73,A -85,B 0,C 180,E1 -15196.074,E2 -15196.074} C_VEL
LIN {X 0,Y 473.646,Z 762.272,A -85,B 0,C 180,E1 -15196.341,E2 -15196.341} C_VEL
LIN {X 0,Y 473.272,Z 772.713,A -85,B 0,C 180,E1 -15196.738,E2 -15196.738} C_VEL
LIN {X 0,Y 472.971,Z 781.546,A -85,B 0,C 180,E1 -15197.165,E2 -15197.165} C_VEL
LIN {X 0,Y 472.492,Z 792.065,A -85,B 0,C 180,E1 -15197.805,E2 -15197.805} C_VEL
LIN {X 0,Y 471.988,Z 801.473,A -85,B 0,C 180,E1 -15198.505,E2 -15198.505} C_VEL
LIN {X 0,Y 471.566,Z 810.35,A -85,B 0,C 180,E1 -15199.3,E2 -15199.3} C_VEL
LIN {X 0,Y 471.15,Z 818.399,A -85,B 0,C 180,E1 -15200.156,E2 -15200.156} C_VEL
LIN {X 0,Y 470.651,Z 826.739,A -85,B 0,C 180,E1 -15201.226,E2 -15201.226} C_VEL
LIN {X 0,Y 470.328,Z 833.687,A -85,B 0,C 180,E1 -15202.297,E2 -15202.297} C_VEL
LIN {X 0,Y 470.15,Z 838.474,A -85,B 0,C 180,E1 -15203.155,E2 -15203.155} C_VEL
LIN {X 0,Y 469.987,Z 844.294,A -85,B 0,C 180,E1 -15204.441,E2 -15204.441} C_VEL
LIN {X 0,Y 469.871,Z 848.841,A -85,B 0,C 180,E1 -15205.726,E2 -15205.726} C_VEL
LIN {X 0,Y 469.812,Z 851.218,A -85,B 0,C 180,E1 -15206.581,E2 -15206.581} C_VEL
LIN {X 0,Y 469.789,Z 854.633,A -85,B 0,C 180,E1 -15208.291,E2 -15208.291} C_VEL
LIN {X 0,Y 469.815,Z 855.614,A -85,B 0,C 180,E1 -15209.146,E2 -15209.146} C_VEL
LIN {X 0,Y 469.778,Z 856.432,A -85,B 0,C 180,E1 -15210.854,E2 -15210.854} C_VEL
LIN {X 0,Y 469.767,Z 855.391,A -85,B 0,C 180,E1 -15212.564,E2 -15212.564} C_VEL
LIN {X 0,Y 469.807,Z 854.339,A -85,B 0,C 180,E1 -15213.419,E2 -15213.419} C_VEL
LIN {X 0,Y 469.96,Z 850.707,A -85,B 0,C 180,E1 -15215.131,E2 -15215.131} C_VEL
LIN {X 0,Y 470.21,Z 846.785,A -85,B 0,C 180,E1 -15216.415,E2 -15216.415} C_VEL
LIN {X 0,Y 470.558,Z 841.704,A -85,B 0,C 180,E1 -15217.699,E2 -15217.699} C_VEL
LIN {X 0,Y 470.998,Z 836.532,A -85,B 0,C 180,E1 -15218.768,E2 -15218.768} C_VEL
LIN {X 0,Y 471.545,Z 830.313,A -85,B 0,C 180,E1 -15219.836,E2 -15219.836} C_VEL
LIN {X 0,Y 472.291,Z 822.83,A -85,B 0,C 180,E1 -15220.9,E2 -15220.9} C_VEL
LIN {X 0,Y 473.089,Z 813.781,A -85,B 0,C 180,E1 -15221.963,E2 -15221.963} C_VEL
LIN {X 0,Y 473.933,Z 805.117,A -85,B 0,C 180,E1 -15222.809,E2 -15222.809} C_VEL
LIN {X 0,Y 474.663,Z 796.11,A -85,B 0,C 180,E1 -15223.548,E2 -15223.548} C_VEL
LIN {X 0,Y 475.353,Z 786.879,A -85,B 0,C 180,E1 -15224.18,E2 -15224.18} C_VEL
LIN {X 0,Y 476.126,Z 775.299,A -85,B 0,C 180,E1 -15224.81,E2 -15224.81} C_VEL
LIN {X 0,Y 476.827,Z 764.747,A -85,B 0,C 180,E1 -15225.251,E2 -15225.251} C_VEL
LIN {X 0,Y 477.414,Z 753.884,A -85,B 0,C 180,E1 -15225.586,E2 -15225.586} C_VEL
LIN {X 0,Y 478.033,Z 732.915,A -85,B 0,C 180,E1 -15226.028,E2 -15226.028} C_VEL
LIN {X 0,Y 479.497,Z 675.491,A -85,B 0,C 180,E1 -15227.186,E2 -15227.186} C_VEL
LIN {X 0,Y 476.919,Z 658.658,A -85,B 0,C 180,E1 -15227.702,E2 -15227.702} C_VEL
LIN {X 0,Y 473.854,Z 644.063,A -85,B 0,C 180,E1 -15228.224,E2 -15228.224} C_VEL
LIN {X 0,Y 475.48,Z 628.746,A -85,B 0,C 180,E1 -15231.383,E2 -15231.383} C_VEL
LIN {X 0,Y 476.333,Z 621.438,A -85,B 0,C 180,E1 -15232.935,E2 -15232.935} C_VEL
LIN {X 0,Y 474.646,Z 611.52,A -85,B 0,C 180,E1 -15235.338,E2 -15235.338} C_VEL
LIN {X 0,Y 472.538,Z 602.053,A -85,B 0,C 180,E1 -15237.835,E2 -15237.835} C_VEL
LIN {X 0,Y 471.704,Z 598.667,A -85,B 0,C 180,E1 -15238.824,E2 -15238.824} C_VEL
LIN {X 0,Y 471.669,Z 598.667,A -85,B 0,C 180,E1 -15241.317,E2 -15241.317} C_VEL
LIN {X 0,Y 471.675,Z 598.663,A -85,B 0,C 180,E1 -15244.354,E2 -15244.354} C_VEL
LIN {X 0,Y 471.668,Z 598.661,A -85,B 0,C 180,E1 -15247.508,E2 -15247.508} C_VEL
LIN {X 0,Y 471.682,Z 598.655,A -85,B 0,C 180,E1 -15249.684,E2 -15249.684} C_VEL
LIN {X 0,Y 471.682,Z 598.66,A -85,B 0,C 180,E1 -15253.086,E2 -15253.086} C_VEL
LIN {X 0,Y 471.701,Z 598.661,A -85,B 0,C 180,E1 -15255.74,E2 -15255.74} C_VEL
LIN {X 0,Y 471.706,Z 598.66,A -85,B 0,C 180,E1 -15259.228,E2 -15259.228} C_VEL
LIN {X 0,Y 471.662,Z 598.665,A -85,B 0,C 180,E1 -15261.914,E2 -15261.914} C_VEL
LIN {X 0,Y 471.697,Z 598.66,A -85,B 0,C 180,E1 -15264.758,E2 -15264.758} C_VEL
LIN {X 0,Y 471.706,Z 598.658,A -85,B 0,C 180,E1 -15267.823,E2 -15267.823} C_VEL
LIN {X 0,Y 471.693,Z 598.664,A -85,B 0,C 180,E1 -15270.657,E2 -15270.657} C_VEL
LIN {X 0,Y 471.704,Z 598.661,A -85,B 0,C 180,E1 -15273.546,E2 -15273.546} C_VEL
LIN {X 0,Y 471.68,Z 598.666,A -85,B 0,C 180,E1 -15276.362,E2 -15276.362} C_VEL
LIN {X 0,Y 471.758,Z 598.658,A -85,B 0,C 180,E1 -15279.293,E2 -15279.293} C_VEL
LIN {X 0,Y 471.762,Z 598.659,A -85,B 0,C 180,E1 -15281.849,E2 -15281.849} C_VEL
LIN {X 0,Y 471.789,Z 598.854,A -85,B 0,C 180,E1 -15284.279,E2 -15284.279} C_VEL
LIN {X 0,Y 473.652,Z 607.153,A -85,B 0,C 180,E1 -15286.749,E2 -15286.749} C_VEL
LIN {X 0,Y 475.393,Z 616.698,A -85,B 0,C 180,E1 -15289.387,E2 -15289.387} C_VEL
LIN {X 0,Y 475.23,Z 621.88,A -85,B 0,C 180,E1 -15290.669,E2 -15290.669} C_VEL
LIN {X 0,Y 474.524,Z 627,A -85,B 0,C 180,E1 -15291.881,E2 -15291.881} C_VEL
LIN {X 0,Y 478.165,Z 641.661,A -85,B 0,C 180,E1 -15292.436,E2 -15292.436} C_VEL
LIN {X 0,Y 480.096,Z 652.978,A -85,B 0,C 180,E1 -15292.794,E2 -15292.794} C_VEL
LIN {X 0,Y 478.073,Z 714.087,A -85,B 0,C 180,E1 -15294.008,E2 -15294.008} C_VEL
LIN {X 0,Y 477.424,Z 735.77,A -85,B 0,C 180,E1 -15294.475,E2 -15294.475} C_VEL
LIN {X 0,Y 476.799,Z 749.58,A -85,B 0,C 180,E1 -15294.943,E2 -15294.943} C_VEL
LIN {X 0,Y 476.101,Z 762.293,A -85,B 0,C 180,E1 -15295.57,E2 -15295.57} C_VEL
LIN {X 0,Y 475.517,Z 772.315,A -85,B 0,C 180,E1 -15296.199,E2 -15296.199} C_VEL
LIN {X 0,Y 474.865,Z 781.891,A -85,B 0,C 180,E1 -15296.935,E2 -15296.935} C_VEL
LIN {X 0,Y 474.149,Z 790.008,A -85,B 0,C 180,E1 -15297.671,E2 -15297.671} C_VEL
LIN {X 0,Y 473.381,Z 797.888,A -85,B 0,C 180,E1 -15298.516,E2 -15298.516} C_VEL
LIN {X 0,Y 472.49,Z 806.096,A -85,B 0,C 180,E1 -15299.575,E2 -15299.575} C_VEL
LIN {X 0,Y 471.788,Z 812.932,A -85,B 0,C 180,E1 -15300.638,E2 -15300.638} C_VEL
LIN {X 0,Y 471.235,Z 818.646,A -85,B 0,C 180,E1 -15301.703,E2 -15301.703} C_VEL
LIN {X 0,Y 470.65,Z 824.189,A -85,B 0,C 180,E1 -15302.986,E2 -15302.986} C_VEL
LIN {X 0,Y 470.406,Z 828.511,A -85,B 0,C 180,E1 -15304.269,E2 -15304.269} C_VEL
LIN {X 0,Y 470.211,Z 830.864,A -85,B 0,C 180,E1 -15305.128,E2 -15305.128} C_VEL
LIN {X 0,Y 469.863,Z 834.028,A -85,B 0,C 180,E1 -15306.849,E2 -15306.849} C_VEL
LIN {X 0,Y 469.724,Z 835.007,A -85,B 0,C 180,E1 -15307.712,E2 -15307.712} C_VEL
LIN {X 0,Y 469.711,Z 835.577,A -85,B 0,C 180,E1 -15309.441,E2 -15309.441} C_VEL
LIN {X 0,Y 469.724,Z 835.201,A -85,B 0,C 180,E1 -15310.308,E2 -15310.308} C_VEL
LIN {X 0,Y 469.662,Z 833.175,A -85,B 0,C 180,E1 -15312.051,E2 -15312.051} C_VEL
LIN {X 0,Y 469.792,Z 830.422,A -85,B 0,C 180,E1 -15313.361,E2 -15313.361} C_VEL
LIN {X 0,Y 469.98,Z 826.535,A -85,B 0,C 180,E1 -15314.676,E2 -15314.676} C_VEL
LIN {X 0,Y 470.171,Z 821.379,A -85,B 0,C 180,E1 -15315.998,E2 -15315.998} C_VEL
LIN {X 0,Y 470.41,Z 816.043,A -85,B 0,C 180,E1 -15317.102,E2 -15317.102} C_VEL
LIN {X 0,Y 470.683,Z 809.535,A -85,B 0,C 180,E1 -15318.21,E2 -15318.21} C_VEL
LIN {X 0,Y 471.113,Z 801.631,A -85,B 0,C 180,E1 -15319.318,E2 -15319.318} C_VEL
LIN {X 0,Y 471.484,Z 794.404,A -85,B 0,C 180,E1 -15320.175,E2 -15320.175} C_VEL
LIN {X 0,Y 471.896,Z 785.081,A -85,B 0,C 180,E1 -15321.097,E2 -15321.097} C_VEL
LIN {X 0,Y 472.408,Z 775.614,A -85,B 0,C 180,E1 -15321.871,E2 -15321.871} C_VEL
LIN {X 0,Y 472.868,Z 765.743,A -85,B 0,C 180,E1 -15322.536,E2 -15322.536} C_VEL
LIN {X 0,Y 473.25,Z 755.536,A -85,B 0,C 180,E1 -15323.092,E2 -15323.092} C_VEL
LIN {X 0,Y 473.516,Z 744.207,A -85,B 0,C 180,E1 -15323.569,E2 -15323.569} C_VEL
LIN {X 0,Y 473.831,Z 733.392,A -85,B 0,C 180,E1 -15323.899,E2 -15323.899} C_VEL
LIN {X 0,Y 474.338,Z 711.233,A -85,B 0,C 180,E1 -15324.335,E2 -15324.335} C_VEL
LIN {X 0,Y 475.365,Z 648.15,A -85,B 0,C 180,E1 -15325.509,E2 -15325.509} C_VEL
LIN {X 0,Y 472.195,Z 624.974,A -85,B 0,C 180,E1 -15326.034,E2 -15326.034} C_VEL
LIN {X 0,Y 473.065,Z 610.629,A -85,B 0,C 180,E1 -15329.122,E2 -15329.122} C_VEL
LIN {X 0,Y 473.116,Z 606.727,A -85,B 0,C 180,E1 -15329.977,E2 -15329.977} C_VEL
LIN {X 0,Y 471.753,Z 598.658,A -85,B 0,C 180,E1 -15331.854,E2 -15331.854} C_VEL
LIN {X 0,Y 471.698,Z 598.66,A -85,B 0,C 180,E1 -15334.352,E2 -15334.352} C_VEL
LIN {X 0,Y 471.67,Z 598.662,A -85,B 0,C 180,E1 -15337.507,E2 -15337.507} C_VEL
LIN {X 0,Y 471.721,Z 598.657,A -85,B 0,C 180,E1 -15339.679,E2 -15339.679} C_VEL
LIN {X 0,Y 471.68,Z 598.658,A -85,B 0,C 180,E1 -15343.086,E2 -15343.086} C_VEL
LIN {X 0,Y 471.7,Z 598.661,A -85,B 0,C 180,E1 -15345.739,E2 -15345.739} C_VEL
LIN {X 0,Y 471.702,Z 598.656,A -85,B 0,C 180,E1 -15349.227,E2 -15349.227} C_VEL
LIN {X 0,Y 471.659,Z 598.668,A -85,B 0,C 180,E1 -15351.913,E2 -15351.913} C_VEL
LIN {X 0,Y 471.694,Z 598.657,A -85,B 0,C 180,E1 -15354.757,E2 -15354.757} C_VEL
LIN {X 0,Y 471.687,Z 598.664,A -85,B 0,C 180,E1 -15357.825,E2 -15357.825} C_VEL
LIN {X 0,Y 471.687,Z 598.658,A -85,B 0,C 180,E1 -15360.656,E2 -15360.656} C_VEL
LIN {X 0,Y 471.697,Z 598.659,A -85,B 0,C 180,E1 -15363.545,E2 -15363.545} C_VEL
LIN {X 0,Y 471.674,Z 598.662,A -85,B 0,C 180,E1 -15366.362,E2 -15366.362} C_VEL
LIN {X 0,Y 471.751,Z 598.65,A -85,B 0,C 180,E1 -15369.292,E2 -15369.292} C_VEL
LIN {X 0,Y 471.727,Z 598.653,A -85,B 0,C 180,E1 -15372.724,E2 -15372.724} C_VEL
LIN {X 0,Y 471.824,Z 598.642,A -85,B 0,C 180,E1 -15375.382,E2 -15375.382} C_VEL
LIN {X 0,Y 471.85,Z 598.637,A -85,B 0,C 180,E1 -15378.873,E2 -15378.873} C_VEL
LIN {X 0,Y 471.884,Z 598.637,A -85,B 0,C 180,E1 -15382.323,E2 -15382.323} C_VEL
LIN {X 0,Y 471.975,Z 598.622,A -85,B 0,C 180,E1 -15384.891,E2 -15384.891} C_VEL
LIN {X 0,Y 471.792,Z 598.646,A -85,B 0,C 180,E1 -15387.447,E2 -15387.447} C_VEL
LIN {X 0,Y 472.041,Z 598.622,A -85,B 0,C 180,E1 -15390,E2 -15390} C_VEL
LIN {X 0,Y 471.967,Z 598.627,A -85,B 0,C 180,E1 -15394.255,E2 -15394.255} C_VEL
LIN {X 0,Y 471.888,Z 598.633,A -85,B 0,C 180,E1 -15396.82,E2 -15396.82} C_VEL
LIN {X 0,Y 471.829,Z 598.641,A -85,B 0,C 180,E1 -15399.398,E2 -15399.398} C_VEL
LIN {X 0,Y 471.82,Z 598.649,A -85,B 0,C 180,E1 -15401.996,E2 -15401.996} C_VEL
LIN {X 0,Y 471.83,Z 598.64,A -85,B 0,C 180,E1 -15405.218,E2 -15405.218} C_VEL
LIN {X 0,Y 471.758,Z 598.654,A -85,B 0,C 180,E1 -15408.167,E2 -15408.167} C_VEL
LIN {X 0,Y 471.724,Z 598.653,A -85,B 0,C 180,E1 -15410.901,E2 -15410.901} C_VEL
LIN {X 0,Y 471.673,Z 598.663,A -85,B 0,C 180,E1 -15413.638,E2 -15413.638} C_VEL
LIN {X 0,Y 471.684,Z 598.659,A -85,B 0,C 180,E1 -15414.618,E2 -15414.618} C_VEL
LIN {X 0,Y 471.02,Z 598.743,A -85,B 0,C 180,E1 -15415.331,E2 -15415.331} C_VEL
LIN {X 0,Y 468.171,Z 599.098,A -85,B 0,C 180,E1 -15416.49,E2 -15416.49} C_VEL
LIN {X 0,Y 465.763,Z 599.399,A -85,B 0,C 180,E1 -15417.424,E2 -15417.424} C_VEL
LIN {X 0,Y 464.733,Z 599.53,A -85,B 0,C 180,E1 -15418.146,E2 -15418.146} C_VEL
LIN {X 0,Y 464.651,Z 599.535,A -85,B 0,C 180,E1 -15418.39,E2 -15418.39} C_VEL
LIN {X 0,Y 464.687,Z 599.53,A -85,B 0,C 180,E1 -15420.83,E2 -15420.83} C_VEL
LIN {X 0,Y 464.687,Z 599.538,A -85,B 0,C 180,E1 -15424.001,E2 -15424.001} C_VEL
LIN {X 0,Y 464.704,Z 599.527,A -85,B 0,C 180,E1 -15427.079,E2 -15427.079} C_VEL
LIN {X 0,Y 464.661,Z 599.536,A -85,B 0,C 180,E1 -15430.406,E2 -15430.406} C_VEL
LIN {X 0,Y 464.643,Z 599.542,A -85,B 0,C 180,E1 -15433.903,E2 -15433.903} C_VEL
LIN {X 0,Y 464.642,Z 599.539,A -85,B 0,C 180,E1 -15436.352,E2 -15436.352} C_VEL
LIN {X 0,Y 464.662,Z 599.536,A -85,B 0,C 180,E1 -15439.595,E2 -15439.595} C_VEL
LIN {X 0,Y 464.689,Z 599.529,A -85,B 0,C 180,E1 -15443.024,E2 -15443.024} C_VEL
LIN {X 0,Y 464.665,Z 599.539,A -85,B 0,C 180,E1 -15446.101,E2 -15446.101} C_VEL
LIN {X 0,Y 464.657,Z 599.534,A -85,B 0,C 180,E1 -15449.232,E2 -15449.232} C_VEL
LIN {X 0,Y 464.675,Z 599.537,A -85,B 0,C 180,E1 -15452.142,E2 -15452.142} C_VEL
LIN {X 0,Y 464.655,Z 599.534,A -85,B 0,C 180,E1 -15455.034,E2 -15455.034} C_VEL
LIN {X 0,Y 464.676,Z 599.537,A -85,B 0,C 180,E1 -15457.862,E2 -15457.862} C_VEL
LIN {X 0,Y 464.678,Z 599.532,A -85,B 0,C 180,E1 -15460.633,E2 -15460.633} C_VEL
LIN {X 0,Y 464.665,Z 599.533,A -85,B 0,C 180,E1 -15463.357,E2 -15463.357} C_VEL
LIN {X 0,Y 464.72,Z 599.533,A -85,B 0,C 180,E1 -15466.045,E2 -15466.045} C_VEL
LIN {X 0,Y 464.799,Z 599.516,A -85,B 0,C 180,E1 -15468.703,E2 -15468.703} C_VEL
LIN {X 0,Y 464.861,Z 599.513,A -85,B 0,C 180,E1 -15472.206,E2 -15472.206} C_VEL
LIN {X 0,Y 464.924,Z 599.5,A -85,B 0,C 180,E1 -15474.814,E2 -15474.814} C_VEL
LIN {X 0,Y 464.77,Z 599.521,A -85,B 0,C 180,E1 -15477.409,E2 -15477.409} C_VEL
LIN {X 0,Y 464.998,Z 599.499,A -85,B 0,C 180,E1 -15480,E2 -15480} C_VEL
LIN {X 0,Y 464.928,Z 599.503,A -85,B 0,C 180,E1 -15484.32,E2 -15484.32} C_VEL
LIN {X 0,Y 464.854,Z 599.509,A -85,B 0,C 180,E1 -15486.924,E2 -15486.924} C_VEL
LIN {X 0,Y 464.779,Z 599.521,A -85,B 0,C 180,E1 -15489.542,E2 -15489.542} C_VEL
LIN {X 0,Y 464.768,Z 599.525,A -85,B 0,C 180,E1 -15492.181,E2 -15492.181} C_VEL
LIN {X 0,Y 464.717,Z 599.526,A -85,B 0,C 180,E1 -15495.283,E2 -15495.283} C_VEL
LIN {X 0,Y 464.67,Z 599.534,A -85,B 0,C 180,E1 -15498.455,E2 -15498.455} C_VEL
LIN {X 0,Y 464.651,Z 599.534,A -85,B 0,C 180,E1 -15501.21,E2 -15501.21} C_VEL
LIN {X 0,Y 464.622,Z 599.546,A -85,B 0,C 180,E1 -15504.019,E2 -15504.019} C_VEL
LIN {X 0,Y 464.665,Z 599.533,A -85,B 0,C 180,E1 -15507.205,E2 -15507.205} C_VEL
LIN {X 0,Y 464.636,Z 599.542,A -85,B 0,C 180,E1 -15509.833,E2 -15509.833} C_VEL
LIN {X 0,Y 464.568,Z 599.544,A -85,B 0,C 180,E1 -15512.873,E2 -15512.873} C_VEL
LIN {X 0,Y 464.636,Z 599.544,A -85,B 0,C 180,E1 -15516.01,E2 -15516.01} C_VEL
LIN {X 0,Y 464.602,Z 599.541,A -85,B 0,C 180,E1 -15519.287,E2 -15519.287} C_VEL
LIN {X 0,Y 464.609,Z 599.542,A -85,B 0,C 180,E1 -15522.377,E2 -15522.377} C_VEL
LIN {X 0,Y 464.667,Z 599.532,A -85,B 0,C 180,E1 -15525.112,E2 -15525.112} C_VEL
LIN {X 0,Y 464.625,Z 599.54,A -85,B 0,C 180,E1 -15528.446,E2 -15528.446} C_VEL
LIN {X 0,Y 464.573,Z 599.55,A -85,B 0,C 180,E1 -15531.818,E2 -15531.818} C_VEL
LIN {X 0,Y 464.619,Z 599.538,A -85,B 0,C 180,E1 -15535.049,E2 -15535.049} C_VEL
LIN {X 0,Y 464.578,Z 599.549,A -85,B 0,C 180,E1 -15538.15,E2 -15538.15} C_VEL
LIN {X 0,Y 464.655,Z 599.534,A -85,B 0,C 180,E1 -15541.159,E2 -15541.159} C_VEL
LIN {X 0,Y 464.663,Z 599.542,A -85,B 0,C 180,E1 -15544.648,E2 -15544.648} C_VEL
LIN {X 0,Y 467.113,Z 613.313,A -85,B 0,C 180,E1 -15547.519,E2 -15547.519} C_VEL
LIN {X 0,Y 466.46,Z 623.724,A -85,B 0,C 180,E1 -15549.566,E2 -15549.566} C_VEL
LIN {X 0,Y 465.127,Z 642.148,A -85,B 0,C 180,E1 -15553.149,E2 -15553.149} C_VEL
LIN {X 0,Y 464.9,Z 645.618,A -85,B 0,C 180,E1 -15553.814,E2 -15553.814} C_VEL
LIN {X 0,Y 468.187,Z 676.501,A -85,B 0,C 180,E1 -15554.497,E2 -15554.497} C_VEL
LIN {X 0,Y 466.83,Z 751.87,A -85,B 0,C 180,E1 -15555.943,E2 -15555.943} C_VEL
LIN {X 0,Y 466.62,Z 762.388,A -85,B 0,C 180,E1 -15556.242,E2 -15556.242} C_VEL
LIN {X 0,Y 466.233,Z 772.743,A -85,B 0,C 180,E1 -15556.645,E2 -15556.645} C_VEL
LIN {X 0,Y 465.934,Z 781.531,A -85,B 0,C 180,E1 -15557.079,E2 -15557.079} C_VEL
LIN {X 0,Y 465.419,Z 792.014,A -85,B 0,C 180,E1 -15557.727,E2 -15557.727} C_VEL
LIN {X 0,Y 464.892,Z 801.82,A -85,B 0,C 180,E1 -15558.474,E2 -15558.474} C_VEL
LIN {X 0,Y 464.505,Z 810.273,A -85,B 0,C 180,E1 -15559.245,E2 -15559.245} C_VEL
LIN {X 0,Y 464.029,Z 819.181,A -85,B 0,C 180,E1 -15560.223,E2 -15560.223} C_VEL
LIN {X 0,Y 463.623,Z 825.92,A -85,B 0,C 180,E1 -15561.092,E2 -15561.092} C_VEL
LIN {X 0,Y 463.263,Z 832.983,A -85,B 0,C 180,E1 -15562.179,E2 -15562.179} C_VEL
LIN {X 0,Y 463.047,Z 838.882,A -85,B 0,C 180,E1 -15563.268,E2 -15563.268} C_VEL
LIN {X 0,Y 462.903,Z 843.772,A -85,B 0,C 180,E1 -15564.356,E2 -15564.356} C_VEL
LIN {X 0,Y 462.781,Z 848.418,A -85,B 0,C 180,E1 -15565.66,E2 -15565.66} C_VEL
LIN {X 0,Y 462.733,Z 850.803,A -85,B 0,C 180,E1 -15566.529,E2 -15566.529} C_VEL
LIN {X 0,Y 462.692,Z 854.357,A -85,B 0,C 180,E1 -15568.265,E2 -15568.265} C_VEL
LIN {X 0,Y 462.708,Z 855.975,A -85,B 0,C 180,E1 -15570,E2 -15570} C_VEL
LIN {X 0,Y 462.689,Z 856.263,A -85,B 0,C 180,E1 -15570.868,E2 -15570.868} C_VEL
LIN {X 0,Y 462.688,Z 855.313,A -85,B 0,C 180,E1 -15572.603,E2 -15572.603} C_VEL
LIN {X 0,Y 462.728,Z 854.264,A -85,B 0,C 180,E1 -15573.472,E2 -15573.472} C_VEL
LIN {X 0,Y 462.883,Z 850.762,A -85,B 0,C 180,E1 -15575.209,E2 -15575.209} C_VEL
LIN {X 0,Y 463.164,Z 846.929,A -85,B 0,C 180,E1 -15576.513,E2 -15576.513} C_VEL
LIN {X 0,Y 463.542,Z 841.936,A -85,B 0,C 180,E1 -15577.816,E2 -15577.816} C_VEL
LIN {X 0,Y 464.059,Z 835.637,A -85,B 0,C 180,E1 -15579.119,E2 -15579.119} C_VEL
LIN {X 0,Y 464.729,Z 829.257,A -85,B 0,C 180,E1 -15580.201,E2 -15580.201} C_VEL
LIN {X 0,Y 465.556,Z 821.591,A -85,B 0,C 180,E1 -15581.279,E2 -15581.279} C_VEL
LIN {X 0,Y 466.173,Z 814.389,A -85,B 0,C 180,E1 -15582.143,E2 -15582.143} C_VEL
LIN {X 0,Y 467.143,Z 804.634,A -85,B 0,C 180,E1 -15583.108,E2 -15583.108} C_VEL
LIN {X 0,Y 467.916,Z 795.578,A -85,B 0,C 180,E1 -15583.858,E2 -15583.858} C_VEL
LIN {X 0,Y 468.687,Z 786.343,A -85,B 0,C 180,E1 -15584.497,E2 -15584.497} C_VEL
LIN {X 0,Y 469.494,Z 774.793,A -85,B 0,C 180,E1 -15585.135,E2 -15585.135} C_VEL
LIN {X 0,Y 470.24,Z 764.256,A -85,B 0,C 180,E1 -15585.58,E2 -15585.58} C_VEL
LIN {X 0,Y 470.855,Z 753.421,A -85,B 0,C 180,E1 -15585.919,E2 -15585.919} C_VEL
LIN {X 0,Y 471.459,Z 733.787,A -85,B 0,C 180,E1 -15586.341,E2 -15586.341} C_VEL
LIN {X 0,Y 473.049,Z 676.616,A -85,B 0,C 180,E1 -15587.516,E2 -15587.516} C_VEL
LIN {X 0,Y 470.908,Z 662.216,A -85,B 0,C 180,E1 -15587.968,E2 -15587.968} C_VEL
LIN {X 0,Y 467.12,Z 644.038,A -85,B 0,C 180,E1 -15588.631,E2 -15588.631} C_VEL
LIN {X 0,Y 468.878,Z 628.307,A -85,B 0,C 180,E1 -15591.93,E2 -15591.93} C_VEL
LIN {X 0,Y 469.483,Z 623.129,A -85,B 0,C 180,E1 -15593.057,E2 -15593.057} C_VEL
LIN {X 0,Y 468.031,Z 614.265,A -85,B 0,C 180,E1 -15595.247,E2 -15595.247} C_VEL
LIN {X 0,Y 465.98,Z 604.853,A -85,B 0,C 180,E1 -15597.774,E2 -15597.774} C_VEL
LIN {X 0,Y 464.643,Z 599.545,A -85,B 0,C 180,E1 -15599.337,E2 -15599.337} C_VEL
LIN {X 0,Y 464.614,Z 599.546,A -85,B 0,C 180,E1 -15602.409,E2 -15602.409} C_VEL
LIN {X 0,Y 464.639,Z 599.54,A -85,B 0,C 180,E1 -15605.506,E2 -15605.506} C_VEL
LIN {X 0,Y 464.614,Z 599.535,A -85,B 0,C 180,E1 -15608.377,E2 -15608.377} C_VEL
LIN {X 0,Y 464.627,Z 599.535,A -85,B 0,C 180,E1 -15611.554,E2 -15611.554} C_VEL
LIN {X 0,Y 464.681,Z 599.534,A -85,B 0,C 180,E1 -15614.89,E2 -15614.89} C_VEL
LIN {X 0,Y 464.645,Z 599.54,A -85,B 0,C 180,E1 -15618.448,E2 -15618.448} C_VEL
LIN {X 0,Y 464.666,Z 599.536,A -85,B 0,C 180,E1 -15620.72,E2 -15620.72} C_VEL
LIN {X 0,Y 464.664,Z 599.536,A -85,B 0,C 180,E1 -15623.992,E2 -15623.992} C_VEL
LIN {X 0,Y 464.656,Z 599.541,A -85,B 0,C 180,E1 -15627.134,E2 -15627.134} C_VEL
LIN {X 0,Y 464.652,Z 599.537,A -85,B 0,C 180,E1 -15630.168,E2 -15630.168} C_VEL
LIN {X 0,Y 464.704,Z 599.532,A -85,B 0,C 180,E1 -15633.116,E2 -15633.116} C_VEL
LIN {X 0,Y 464.626,Z 599.542,A -85,B 0,C 180,E1 -15635.981,E2 -15635.981} C_VEL
LIN {X 0,Y 464.704,Z 599.538,A -85,B 0,C 180,E1 -15639.152,E2 -15639.152} C_VEL
LIN {X 0,Y 464.69,Z 599.54,A -85,B 0,C 180,E1 -15642.454,E2 -15642.454} C_VEL
LIN {X 0,Y 464.705,Z 599.671,A -85,B 0,C 180,E1 -15643.752,E2 -15643.752} C_VEL
LIN {X 0,Y 466.492,Z 607.232,A -85,B 0,C 180,E1 -15646.099,E2 -15646.099} C_VEL
LIN {X 0,Y 468.289,Z 616.636,A -85,B 0,C 180,E1 -15648.787,E2 -15648.787} C_VEL
LIN {X 0,Y 468.563,Z 621.618,A -85,B 0,C 180,E1 -15650.101,E2 -15650.101} C_VEL
LIN {X 0,Y 467.864,Z 627.219,A -85,B 0,C 180,E1 -15651.461,E2 -15651.461} C_VEL
LIN {X 0,Y 471.696,Z 642.772,A -85,B 0,C 180,E1 -15652.078,E2 -15652.078} C_VEL
LIN {X 0,Y 473.666,Z 654.089,A -85,B 0,C 180,E1 -15652.457,E2 -15652.457} C_VEL
LIN {X 0,Y 471.529,Z 714.744,A -85,B 0,C 180,E1 -15653.683,E2 -15653.683} C_VEL
LIN {X 0,Y 470.856,Z 736.217,A -85,B 0,C 180,E1 -15654.157,E2 -15654.157} C_VEL
LIN {X 0,Y 470.176,Z 750.454,A -85,B 0,C 180,E1 -15654.657,E2 -15654.657} C_VEL
LIN {X 0,Y 469.54,Z 761.198,A -85,B 0,C 180,E1 -15655.186,E2 -15655.186} C_VEL
LIN {X 0,Y 468.798,Z 772.836,A -85,B 0,C 180,E1 -15655.93,E2 -15655.93} C_VEL
LIN {X 0,Y 468.094,Z 782.307,A -85,B 0,C 180,E1 -15656.676,E2 -15656.676} C_VEL
LIN {X 0,Y 467.239,Z 791.371,A -85,B 0,C 180,E1 -15657.53,E2 -15657.53} C_VEL
LIN {X 0,Y 466.546,Z 798.212,A -85,B 0,C 180,E1 -15658.279,E2 -15658.279} C_VEL
LIN {X 0,Y 465.629,Z 806.403,A -85,B 0,C 180,E1 -15659.353,E2 -15659.353} C_VEL
LIN {X 0,Y 464.857,Z 813.234,A -85,B 0,C 180,E1 -15660.431,E2 -15660.431} C_VEL
LIN {X 0,Y 464.416,Z 817.935,A -85,B 0,C 180,E1 -15661.296,E2 -15661.296} C_VEL
LIN {X 0,Y 463.702,Z 823.697,A -85,B 0,C 180,E1 -15662.597,E2 -15662.597} C_VEL
LIN {X 0,Y 463.429,Z 828.47,A -85,B 0,C 180,E1 -15664.008,E2 -15664.008} C_VEL
LIN {X 0,Y 463.105,Z 831.595,A -85,B 0,C 180,E1 -15665.206,E2 -15665.206} C_VEL
LIN {X 0,Y 462.923,Z 833.242,A -85,B 0,C 180,E1 -15666.08,E2 -15666.08} C_VEL
LIN {X 0,Y 462.624,Z 835.387,A -85,B 0,C 180,E1 -15667.832,E2 -15667.832} C_VEL
LIN {X 0,Y 462.62,Z 835.647,A -85,B 0,C 180,E1 -15669.587,E2 -15669.587} C_VEL
LIN {X 0,Y 462.623,Z 835.25,A -85,B 0,C 180,E1 -15670.468,E2 -15670.468} C_VEL
LIN {X 0,Y 462.566,Z 832.861,A -85,B 0,C 180,E1 -15672.239,E2 -15672.239} C_VEL
LIN {X 0,Y 462.725,Z 829.903,A -85,B 0,C 180,E1 -15673.569,E2 -15673.569} C_VEL
LIN {X 0,Y 462.898,Z 827.464,A -85,B 0,C 180,E1 -15674.434,E2 -15674.434} C_VEL
LIN {X 0,Y 463.102,Z 821.415,A -85,B 0,C 180,E1 -15676.023,E2 -15676.023} C_VEL
LIN {X 0,Y 463.32,Z 816.036,A -85,B 0,C 180,E1 -15677.145,E2 -15677.145} C_VEL
LIN {X 0,Y 463.62,Z 809.318,A -85,B 0,C 180,E1 -15678.295,E2 -15678.295} C_VEL
LIN {X 0,Y 464.037,Z 801.527,A -85,B 0,C 180,E1 -15679.395,E2 -15679.395} C_VEL
LIN {X 0,Y 464.433,Z 793.942,A -85,B 0,C 180,E1 -15680.296,E2 -15680.296} C_VEL
LIN {X 0,Y 464.844,Z 784.845,A -85,B 0,C 180,E1 -15681.201,E2 -15681.201} C_VEL
LIN {X 0,Y 465.387,Z 775.299,A -85,B 0,C 180,E1 -15681.986,E2 -15681.986} C_VEL
LIN {X 0,Y 465.822,Z 765.294,A -85,B 0,C 180,E1 -15682.663,E2 -15682.663} C_VEL
LIN {X 0,Y 466.266,Z 754.805,A -85,B 0,C 180,E1 -15683.232,E2 -15683.232} C_VEL
LIN {X 0,Y 466.495,Z 744.174,A -85,B 0,C 180,E1 -15683.682,E2 -15683.682} C_VEL
LIN {X 0,Y 466.805,Z 733.323,A -85,B 0,C 180,E1 -15684.017,E2 -15684.017} C_VEL
LIN {X 0,Y 467.291,Z 712.674,A -85,B 0,C 180,E1 -15684.432,E2 -15684.432} C_VEL
LIN {X 0,Y 468.347,Z 648.743,A -85,B 0,C 180,E1 -15685.653,E2 -15685.653} C_VEL
LIN {X 0,Y 465.178,Z 625.085,A -85,B 0,C 180,E1 -15686.21,E2 -15686.21} C_VEL
LIN {X 0,Y 466.099,Z 610.672,A -85,B 0,C 180,E1 -15689.353,E2 -15689.353} C_VEL
LIN {X 0,Y 465.947,Z 606.723,A -85,B 0,C 180,E1 -15690.238,E2 -15690.238} C_VEL
LIN {X 0,Y 464.691,Z 599.537,A -85,B 0,C 180,E1 -15691.941,E2 -15691.941} C_VEL
LIN {X 0,Y 464.649,Z 599.534,A -85,B 0,C 180,E1 -15694.948,E2 -15694.948} C_VEL
LIN {X 0,Y 464.614,Z 599.544,A -85,B 0,C 180,E1 -15698.178,E2 -15698.178} C_VEL
LIN {X 0,Y 464.662,Z 599.536,A -85,B 0,C 180,E1 -15700.405,E2 -15700.405} C_VEL
LIN {X 0,Y 464.646,Z 599.542,A -85,B 0,C 180,E1 -15703.902,E2 -15703.902} C_VEL
LIN {X 0,Y 464.643,Z 599.538,A -85,B 0,C 180,E1 -15706.351,E2 -15706.351} C_VEL
LIN {X 0,Y 464.661,Z 599.536,A -85,B 0,C 180,E1 -15709.594,E2 -15709.594} C_VEL
LIN {X 0,Y 464.631,Z 599.536,A -85,B 0,C 180,E1 -15713.033,E2 -15713.033} C_VEL
LIN {X 0,Y 464.665,Z 599.539,A -85,B 0,C 180,E1 -15716.1,E2 -15716.1} C_VEL
LIN {X 0,Y 464.655,Z 599.534,A -85,B 0,C 180,E1 -15719.231,E2 -15719.231} C_VEL
LIN {X 0,Y 464.673,Z 599.537,A -85,B 0,C 180,E1 -15722.141,E2 -15722.141} C_VEL
LIN {X 0,Y 464.653,Z 599.534,A -85,B 0,C 180,E1 -15725.033,E2 -15725.033} C_VEL
LIN {X 0,Y 464.674,Z 599.538,A -85,B 0,C 180,E1 -15727.861,E2 -15727.861} C_VEL
LIN {X 0,Y 464.677,Z 599.532,A -85,B 0,C 180,E1 -15730.632,E2 -15730.632} C_VEL
LIN {X 0,Y 464.694,Z 599.53,A -85,B 0,C 180,E1 -15733.358,E2 -15733.358} C_VEL
LIN {X 0,Y 464.746,Z 599.53,A -85,B 0,C 180,E1 -15736.046,E2 -15736.046} C_VEL
LIN {X 0,Y 464.796,Z 599.517,A -85,B 0,C 180,E1 -15738.702,E2 -15738.702} C_VEL
LIN {X 0,Y 464.856,Z 599.514,A -85,B 0,C 180,E1 -15742.206,E2 -15742.206} C_VEL
LIN {X 0,Y 464.922,Z 599.5,A -85,B 0,C 180,E1 -15744.813,E2 -15744.813} C_VEL
LIN {X 0,Y 464.768,Z 599.521,A -85,B 0,C 180,E1 -15747.408,E2 -15747.408} C_VEL
LIN {X 0,Y 464.995,Z 599.499,A -85,B 0,C 180,E1 -15750,E2 -15750} C_VEL
LIN {X 0,Y 464.936,Z 599.502,A -85,B 0,C 180,E1 -15754.32,E2 -15754.32} C_VEL
LIN {X 0,Y 464.849,Z 599.509,A -85,B 0,C 180,E1 -15756.923,E2 -15756.923} C_VEL
LIN {X 0,Y 464.773,Z 599.521,A -85,B 0,C 180,E1 -15759.542,E2 -15759.542} C_VEL
LIN {X 0,Y 464.77,Z 599.525,A -85,B 0,C 180,E1 -15762.18,E2 -15762.18} C_VEL
LIN {X 0,Y 464.772,Z 599.52,A -85,B 0,C 180,E1 -15765.309,E2 -15765.309} C_VEL
LIN {X 0,Y 464.705,Z 599.53,A -85,B 0,C 180,E1 -15768.453,E2 -15768.453} C_VEL
LIN {X 0,Y 464.671,Z 599.532,A -85,B 0,C 180,E1 -15771.209,E2 -15771.209} C_VEL
LIN {X 0,Y 464.619,Z 599.546,A -85,B 0,C 180,E1 -15774.019,E2 -15774.019} C_VEL
LIN {X 0,Y 464.668,Z 599.532,A -85,B 0,C 180,E1 -15777.207,E2 -15777.207} C_VEL
LIN {X 0,Y 464.651,Z 599.535,A -85,B 0,C 180,E1 -15778.39,E2 -15778.39} C_VEL
LIN {X 0,Y 463.982,Z 599.618,A -85,B 0,C 180,E1 -15779.114,E2 -15779.114} C_VEL
LIN {X 0,Y 461.104,Z 599.98,A -85,B 0,C 180,E1 -15780.29,E2 -15780.29} C_VEL
LIN {X 0,Y 458.689,Z 600.277,A -85,B 0,C 180,E1 -15781.238,E2 -15781.238} C_VEL
LIN {X 0,Y 457.682,Z 600.41,A -85,B 0,C 180,E1 -15781.971,E2 -15781.971} C_VEL
LIN {X 0,Y 457.616,Z 600.412,A -85,B 0,C 180,E1 -15782.219,E2 -15782.219} C_VEL
LIN {X 0,Y 457.647,Z 600.409,A -85,B 0,C 180,E1 -15785.563,E2 -15785.563} C_VEL
LIN {X 0,Y 457.6,Z 600.413,A -85,B 0,C 180,E1 -15788.681,E2 -15788.681} C_VEL
LIN {X 0,Y 457.603,Z 600.413,A -85,B 0,C 180,E1 -15791.408,E2 -15791.408} C_VEL
LIN {X 0,Y 457.639,Z 600.408,A -85,B 0,C 180,E1 -15794.753,E2 -15794.753} C_VEL
LIN {X 0,Y 457.606,Z 600.415,A -85,B 0,C 180,E1 -15797.663,E2 -15797.663} C_VEL
LIN {X 0,Y 457.646,Z 600.415,A -85,B 0,C 180,E1 -15799.998,E2 -15799.998} C_VEL
LIN {X 0,Y 457.637,Z 600.409,A -85,B 0,C 180,E1 -15803.351,E2 -15803.351} C_VEL
LIN {X 0,Y 457.613,Z 600.412,A -85,B 0,C 180,E1 -15806.563,E2 -15806.563} C_VEL
LIN {X 0,Y 457.613,Z 600.415,A -85,B 0,C 180,E1 -15809.662,E2 -15809.662} C_VEL
LIN {X 0,Y 457.636,Z 600.409,A -85,B 0,C 180,E1 -15812.667,E2 -15812.667} C_VEL
LIN {X 0,Y 457.584,Z 600.417,A -85,B 0,C 180,E1 -15815.588,E2 -15815.588} C_VEL
LIN {X 0,Y 457.656,Z 600.405,A -85,B 0,C 180,E1 -15819.004,E2 -15819.004} C_VEL
LIN {X 0,Y 457.655,Z 600.411,A -85,B 0,C 180,E1 -15822.176,E2 -15822.176} C_VEL
LIN {X 0,Y 457.705,Z 600.399,A -85,B 0,C 180,E1 -15824.921,E2 -15824.921} C_VEL
LIN {X 0,Y 457.758,Z 600.395,A -85,B 0,C 180,E1 -15828.526,E2 -15828.526} C_VEL
LIN {X 0,Y 457.812,Z 600.393,A -85,B 0,C 180,E1 -15832.086,E2 -15832.086} C_VEL
LIN {X 0,Y 457.879,Z 600.378,A -85,B 0,C 180,E1 -15834.734,E2 -15834.734} C_VEL
LIN {X 0,Y 457.747,Z 600.395,A -85,B 0,C 180,E1 -15837.369,E2 -15837.369} C_VEL
LIN {X 0,Y 457.951,Z 600.377,A -85,B 0,C 180,E1 -15840,E2 -15840} C_VEL
LIN {X 0,Y 457.897,Z 600.378,A -85,B 0,C 180,E1 -15844.387,E2 -15844.387} C_VEL
LIN {X 0,Y 457.823,Z 600.385,A -85,B 0,C 180,E1 -15847.031,E2 -15847.031} C_VEL
LIN {X 0,Y 457.728,Z 600.401,A -85,B 0,C 180,E1 -15849.691,E2 -15849.691} C_VEL
LIN {X 0,Y 457.709,Z 600.402,A -85,B 0,C 180,E1 -15852.371,E2 -15852.371} C_VEL
LIN {X 0,Y 457.675,Z 600.404,A -85,B 0,C 180,E1 -15855.383,E2 -15855.383} C_VEL
LIN {X 0,Y 457.621,Z 600.41,A -85,B 0,C 180,E1 -15858.75,E2 -15858.75} C_VEL
LIN {X 0,Y 457.592,Z 600.416,A -85,B 0,C 180,E1 -15861.554,E2 -15861.554} C_VEL
LIN {X 0,Y 457.584,Z 600.417,A -85,B 0,C 180,E1 -15864.413,E2 -15864.413} C_VEL
LIN {X 0,Y 457.621,Z 600.411,A -85,B 0,C 180,E1 -15867.407,E2 -15867.407} C_VEL
LIN {X 0,Y 457.582,Z 600.418,A -85,B 0,C 180,E1 -15870.341,E2 -15870.341} C_VEL
LIN {X 0,Y 457.562,Z 600.419,A -85,B 0,C 180,E1 -15873.442,E2 -15873.442} C_VEL
LIN {X 0,Y 457.575,Z 600.417,A -85,B 0,C 180,E1 -15876.656,E2 -15876.656} C_VEL
LIN {X 0,Y 457.55,Z 600.426,A -85,B 0,C 180,E1 -15880.055,E2 -15880.055} C_VEL
LIN {X 0,Y 457.573,Z 600.416,A -85,B 0,C 180,E1 -15882.712,E2 -15882.712} C_VEL
LIN {X 0,Y 457.61,Z 600.412,A -85,B 0,C 180,E1 -15885.243,E2 -15885.243} C_VEL
LIN {X 0,Y 457.586,Z 600.416,A -85,B 0,C 180,E1 -15888.596,E2 -15888.596} C_VEL
LIN {X 0,Y 457.551,Z 600.419,A -85,B 0,C 180,E1 -15891.328,E2 -15891.328} C_VEL
LIN {X 0,Y 457.564,Z 600.42,A -85,B 0,C 180,E1 -15894.429,E2 -15894.429} C_VEL
LIN {X 0,Y 457.564,Z 600.42,A -85,B 0,C 180,E1 -15897.603,E2 -15897.603} C_VEL
LIN {X 0,Y 457.627,Z 600.41,A -85,B 0,C 180,E1 -15900.744,E2 -15900.744} C_VEL
LIN {X 0,Y 457.63,Z 600.417,A -85,B 0,C 180,E1 -15904.138,E2 -15904.138} C_VEL
LIN {X 0,Y 457.658,Z 600.502,A -85,B 0,C 180,E1 -15904.554,E2 -15904.554} C_VEL
LIN {X 0,Y 460.053,Z 613.881,A -85,B 0,C 180,E1 -15907.391,E2 -15907.391} C_VEL
LIN {X 0,Y 459.653,Z 621.993,A -85,B 0,C 180,E1 -15909.016,E2 -15909.016} C_VEL
LIN {X 0,Y 458.29,Z 639.25,A -85,B 0,C 180,E1 -15912.431,E2 -15912.431} C_VEL
LIN {X 0,Y 457.911,Z 645.368,A -85,B 0,C 180,E1 -15913.633,E2 -15913.633} C_VEL
LIN {X 0,Y 460.825,Z 672.458,A -85,B 0,C 180,E1 -15914.264,E2 -15914.264} C_VEL
LIN {X 0,Y 461.178,Z 678.52,A -85,B 0,C 180,E1 -15914.393,E2 -15914.393} C_VEL
LIN {X 0,Y 459.799,Z 752.137,A -85,B 0,C 180,E1 -15915.837,E2 -15915.837} C_VEL
LIN {X 0,Y 459.589,Z 762.501,A -85,B 0,C 180,E1 -15916.139,E2 -15916.139} C_VEL
LIN {X 0,Y 459.189,Z 772.771,A -85,B 0,C 180,E1 -15916.549,E2 -15916.549} C_VEL
LIN {X 0,Y 458.894,Z 781.514,A -85,B 0,C 180,E1 -15916.989,E2 -15916.989} C_VEL
LIN {X 0,Y 458.358,Z 791.965,A -85,B 0,C 180,E1 -15917.647,E2 -15917.647} C_VEL
LIN {X 0,Y 457.903,Z 800.515,A -85,B 0,C 180,E1 -15918.296,E2 -15918.296} C_VEL
LIN {X 0,Y 457.443,Z 810.196,A -85,B 0,C 180,E1 -15919.189,E2 -15919.189} C_VEL
LIN {X 0,Y 456.983,Z 818.223,A -85,B 0,C 180,E1 -15920.071,E2 -15920.071} C_VEL
LIN {X 0,Y 456.496,Z 826.552,A -85,B 0,C 180,E1 -15921.174,E2 -15921.174} C_VEL
LIN {X 0,Y 456.154,Z 833.487,A -85,B 0,C 180,E1 -15922.279,E2 -15922.279} C_VEL
LIN {X 0,Y 455.933,Z 839.268,A -85,B 0,C 180,E1 -15923.384,E2 -15923.384} C_VEL
LIN {X 0,Y 455.834,Z 843.219,A -85,B 0,C 180,E1 -15924.268,E2 -15924.268} C_VEL
LIN {X 0,Y 455.7,Z 847.97,A -85,B 0,C 180,E1 -15925.592,E2 -15925.592} C_VEL
LIN {X 0,Y 455.636,Z 851.549,A -85,B 0,C 180,E1 -15926.916,E2 -15926.916} C_VEL
LIN {X 0,Y 455.612,Z 854.06,A -85,B 0,C 180,E1 -15928.238,E2 -15928.238} C_VEL
LIN {X 0,Y 455.62,Z 855.774,A -85,B 0,C 180,E1 -15930,E2 -15930} C_VEL
LIN {X 0,Y 455.602,Z 856.073,A -85,B 0,C 180,E1 -15930.881,E2 -15930.881} C_VEL
LIN {X 0,Y 455.591,Z 855.251,A -85,B 0,C 180,E1 -15932.644,E2 -15932.644} C_VEL
LIN {X 0,Y 455.631,Z 854.205,A -85,B 0,C 180,E1 -15933.526,E2 -15933.526} C_VEL
LIN {X 0,Y 455.824,Z 850.849,A -85,B 0,C 180,E1 -15935.29,E2 -15935.29} C_VEL
LIN {X 0,Y 456.094,Z 847.088,A -85,B 0,C 180,E1 -15936.614,E2 -15936.614} C_VEL
LIN {X 0,Y 456.511,Z 842.168,A -85,B 0,C 180,E1 -15937.938,E2 -15937.938} C_VEL
LIN {X 0,Y 457.072,Z 835.947,A -85,B 0,C 180,E1 -15939.26,E2 -15939.26} C_VEL
LIN {X 0,Y 457.766,Z 829.652,A -85,B 0,C 180,E1 -15940.358,E2 -15940.358} C_VEL
LIN {X 0,Y 458.631,Z 822.091,A -85,B 0,C 180,E1 -15941.452,E2 -15941.452} C_VEL
LIN {X 0,Y 459.49,Z 813.278,A -85,B 0,C 180,E1 -15942.518,E2 -15942.518} C_VEL
LIN {X 0,Y 460.408,Z 804.325,A -85,B 0,C 180,E1 -15943.415,E2 -15943.415} C_VEL
LIN {X 0,Y 461.236,Z 795.289,A -85,B 0,C 180,E1 -15944.175,E2 -15944.175} C_VEL
LIN {X 0,Y 462.032,Z 786.026,A -85,B 0,C 180,E1 -15944.823,E2 -15944.823} C_VEL
LIN {X 0,Y 462.823,Z 775.571,A -85,B 0,C 180,E1 -15945.414,E2 -15945.414} C_VEL
LIN {X 0,Y 463.68,Z 763.852,A -85,B 0,C 180,E1 -15945.919,E2 -15945.919} C_VEL
LIN {X 0,Y 464.276,Z 754.031,A -85,B 0,C 180,E1 -15946.235,E2 -15946.235} C_VEL
LIN {X 0,Y 464.848,Z 736.048,A -85,B 0,C 180,E1 -15946.637,E2 -15946.637} C_VEL
LIN {X 0,Y 466.628,Z 677.503,A -85,B 0,C 180,E1 -15947.867,E2 -15947.867} C_VEL
LIN {X 0,Y 464.301,Z 661.888,A -85,B 0,C 180,E1 -15948.384,E2 -15948.384} C_VEL
LIN {X 0,Y 460.754,Z 645.665,A -85,B 0,C 180,E1 -15949.007,E2 -15949.007} C_VEL
LIN {X 0,Y 460.361,Z 643.636,A -85,B 0,C 180,E1 -15949.1,E2 -15949.1} C_VEL
LIN {X 0,Y 462.317,Z 628.097,A -85,B 0,C 180,E1 -15952.453,E2 -15952.453} C_VEL
LIN {X 0,Y 462.653,Z 624.82,A -85,B 0,C 180,E1 -15953.181,E2 -15953.181} C_VEL
LIN {X 0,Y 461.017,Z 615.093,A -85,B 0,C 180,E1 -15955.659,E2 -15955.659} C_VEL
LIN {X 0,Y 458.987,Z 605.837,A -85,B 0,C 180,E1 -15958.235,E2 -15958.235} C_VEL
LIN {X 0,Y 457.602,Z 600.422,A -85,B 0,C 180,E1 -15959.896,E2 -15959.896} C_VEL
LIN {X 0,Y 457.587,Z 600.421,A -85,B 0,C 180,E1 -15963.44,E2 -15963.44} C_VEL
LIN {X 0,Y 457.595,Z 600.414,A -85,B 0,C 180,E1 -15966.654,E2 -15966.654} C_VEL
LIN {X 0,Y 457.582,Z 600.411,A -85,B 0,C 180,E1 -15970.06,E2 -15970.06} C_VEL
LIN {X 0,Y 457.601,Z 600.412,A -85,B 0,C 180,E1 -15973.536,E2 -15973.536} C_VEL
LIN {X 0,Y 457.602,Z 600.417,A -85,B 0,C 180,E1 -15976.464,E2 -15976.464} C_VEL
LIN {X 0,Y 457.651,Z 600.411,A -85,B 0,C 180,E1 -15979.998,E2 -15979.998} C_VEL
LIN {X 0,Y 457.597,Z 600.42,A -85,B 0,C 180,E1 -15983.346,E2 -15983.346} C_VEL
LIN {X 0,Y 457.621,Z 600.413,A -85,B 0,C 180,E1 -15986.563,E2 -15986.563} C_VEL
LIN {X 0,Y 457.618,Z 600.412,A -85,B 0,C 180,E1 -15989.661,E2 -15989.661} C_VEL
LIN {X 0,Y 457.658,Z 600.411,A -85,B 0,C 180,E1 -15992.668,E2 -15992.668} C_VEL
LIN {X 0,Y 457.588,Z 600.419,A -85,B 0,C 180,E1 -15995.588,E2 -15995.588} C_VEL
LIN {X 0,Y 457.661,Z 600.417,A -85,B 0,C 180,E1 -15999.004,E2 -15999.004} C_VEL
LIN {X 0,Y 457.659,Z 600.418,A -85,B 0,C 180,E1 -16002.176,E2 -16002.176} C_VEL
LIN {X 0,Y 457.64,Z 600.563,A -85,B 0,C 180,E1 -16003.208,E2 -16003.208} C_VEL
LIN {X 0,Y 459.649,Z 608.908,A -85,B 0,C 180,E1 -16005.888,E2 -16005.888} C_VEL
LIN {X 0,Y 461.427,Z 618.212,A -85,B 0,C 180,E1 -16008.618,E2 -16008.618} C_VEL
LIN {X 0,Y 461.739,Z 623.178,A -85,B 0,C 180,E1 -16009.953,E2 -16009.953} C_VEL
LIN {X 0,Y 461.21,Z 627.422,A -85,B 0,C 180,E1 -16011.016,E2 -16011.016} C_VEL
LIN {X 0,Y 465.32,Z 643.859,A -85,B 0,C 180,E1 -16011.702,E2 -16011.702} C_VEL
LIN {X 0,Y 467.223,Z 654.322,A -85,B 0,C 180,E1 -16012.071,E2 -16012.071} C_VEL
LIN {X 0,Y 465.154,Z 711.35,A -85,B 0,C 180,E1 -16013.271,E2 -16013.271} C_VEL
LIN {X 0,Y 464.388,Z 734.552,A -85,B 0,C 180,E1 -16013.776,E2 -16013.776} C_VEL
LIN {X 0,Y 463.87,Z 745.357,A -85,B 0,C 180,E1 -16014.123,E2 -16014.123} C_VEL
LIN {X 0,Y 463.206,Z 756.92,A -85,B 0,C 180,E1 -16014.631,E2 -16014.631} C_VEL
LIN {X 0,Y 462.442,Z 768.993,A -85,B 0,C 180,E1 -16015.33,E2 -16015.33} C_VEL
LIN {X 0,Y 461.452,Z 781.685,A -85,B 0,C 180,E1 -16016.301,E2 -16016.301} C_VEL
LIN {X 0,Y 460.581,Z 790.86,A -85,B 0,C 180,E1 -16017.167,E2 -16017.167} C_VEL
LIN {X 0,Y 459.734,Z 798.637,A -85,B 0,C 180,E1 -16018.035,E2 -16018.035} C_VEL
LIN {X 0,Y 458.776,Z 806.754,A -85,B 0,C 180,E1 -16019.125,E2 -16019.125} C_VEL
LIN {X 0,Y 457.941,Z 813.539,A -85,B 0,C 180,E1 -16020.219,E2 -16020.219} C_VEL
LIN {X 0,Y 457.348,Z 819.216,A -85,B 0,C 180,E1 -16021.316,E2 -16021.316} C_VEL
LIN {X 0,Y 456.623,Z 824.74,A -85,B 0,C 180,E1 -16022.637,E2 -16022.637} C_VEL
LIN {X 0,Y 456.371,Z 828.976,A -85,B 0,C 180,E1 -16023.943,E2 -16023.943} C_VEL
LIN {X 0,Y 456.02,Z 832.241,A -85,B 0,C 180,E1 -16025.288,E2 -16025.288} C_VEL
LIN {X 0,Y 455.829,Z 833.889,A -85,B 0,C 180,E1 -16026.175,E2 -16026.175} C_VEL
LIN {X 0,Y 455.535,Z 835.659,A -85,B 0,C 180,E1 -16027.954,E2 -16027.954} C_VEL
LIN {X 0,Y 455.517,Z 835.957,A -85,B 0,C 180,E1 -16028.845,E2 -16028.845} C_VEL
LIN {X 0,Y 455.53,Z 835.161,A -85,B 0,C 180,E1 -16030.633,E2 -16030.633} C_VEL
LIN {X 0,Y 455.481,Z 834.1,A -85,B 0,C 180,E1 -16031.532,E2 -16031.532} C_VEL
LIN {X 0,Y 455.616,Z 830.615,A -85,B 0,C 180,E1 -16033.332,E2 -16033.332} C_VEL
LIN {X 0,Y 455.805,Z 826.417,A -85,B 0,C 180,E1 -16034.758,E2 -16034.758} C_VEL
LIN {X 0,Y 456.015,Z 821.445,A -85,B 0,C 180,E1 -16036.05,E2 -16036.05} C_VEL
LIN {X 0,Y 456.23,Z 816.028,A -85,B 0,C 180,E1 -16037.19,E2 -16037.19} C_VEL
LIN {X 0,Y 456.539,Z 809.438,A -85,B 0,C 180,E1 -16038.331,E2 -16038.331} C_VEL
LIN {X 0,Y 456.977,Z 801.423,A -85,B 0,C 180,E1 -16039.474,E2 -16039.474} C_VEL
LIN {X 0,Y 457.367,Z 793.776,A -85,B 0,C 180,E1 -16040.39,E2 -16040.39} C_VEL
LIN {X 0,Y 457.784,Z 785.061,A -85,B 0,C 180,E1 -16041.268,E2 -16041.268} C_VEL
LIN {X 0,Y 458.354,Z 774.977,A -85,B 0,C 180,E1 -16042.105,E2 -16042.105} C_VEL
LIN {X 0,Y 458.745,Z 766.798,A -85,B 0,C 180,E1 -16042.677,E2 -16042.677} C_VEL
LIN {X 0,Y 459.19,Z 755.582,A -85,B 0,C 180,E1 -16043.306,E2 -16043.306} C_VEL
LIN {X 0,Y 459.435,Z 744.671,A -85,B 0,C 180,E1 -16043.78,E2 -16043.78} C_VEL
LIN {X 0,Y 459.78,Z 733.656,A -85,B 0,C 180,E1 -16044.128,E2 -16044.128} C_VEL
LIN {X 0,Y 460.285,Z 712.71,A -85,B 0,C 180,E1 -16044.559,E2 -16044.559} C_VEL
LIN {X 0,Y 461.365,Z 649.441,A -85,B 0,C 180,E1 -16045.791,E2 -16045.791} C_VEL
LIN {X 0,Y 458.158,Z 625.202,A -85,B 0,C 180,E1 -16046.379,E2 -16046.379} C_VEL
LIN {X 0,Y 459.007,Z 612.321,A -85,B 0,C 180,E1 -16049.23,E2 -16049.23} C_VEL
LIN {X 0,Y 458.962,Z 607.849,A -85,B 0,C 180,E1 -16050.24,E2 -16050.24} C_VEL
LIN {X 0,Y 457.665,Z 600.412,A -85,B 0,C 180,E1 -16052,E2 -16052} C_VEL
LIN {X 0,Y 457.609,Z 600.414,A -85,B 0,C 180,E1 -16055.566,E2 -16055.566} C_VEL
LIN {X 0,Y 457.593,Z 600.413,A -85,B 0,C 180,E1 -16058.872,E2 -16058.872} C_VEL
LIN {X 0,Y 457.606,Z 600.413,A -85,B 0,C 180,E1 -16061.407,E2 -16061.407} C_VEL
LIN {X 0,Y 457.641,Z 600.408,A -85,B 0,C 180,E1 -16064.752,E2 -16064.752} C_VEL
LIN {X 0,Y 457.607,Z 600.415,A -85,B 0,C 180,E1 -16067.662,E2 -16067.662} C_VEL
LIN {X 0,Y 457.647,Z 600.415,A -85,B 0,C 180,E1 -16069.997,E2 -16069.997} C_VEL
LIN {X 0,Y 457.593,Z 600.414,A -85,B 0,C 180,E1 -16073.346,E2 -16073.346} C_VEL
LIN {X 0,Y 457.612,Z 600.412,A -85,B 0,C 180,E1 -16076.562,E2 -16076.562} C_VEL
LIN {X 0,Y 457.611,Z 600.415,A -85,B 0,C 180,E1 -16079.661,E2 -16079.661} C_VEL
LIN {X 0,Y 457.635,Z 600.409,A -85,B 0,C 180,E1 -16082.666,E2 -16082.666} C_VEL
LIN {X 0,Y 457.582,Z 600.417,A -85,B 0,C 180,E1 -16085.587,E2 -16085.587} C_VEL
LIN {X 0,Y 457.654,Z 600.406,A -85,B 0,C 180,E1 -16089.003,E2 -16089.003} C_VEL
LIN {X 0,Y 457.661,Z 600.41,A -85,B 0,C 180,E1 -16092.176,E2 -16092.176} C_VEL
LIN {X 0,Y 457.751,Z 600.394,A -85,B 0,C 180,E1 -16094.922,E2 -16094.922} C_VEL
LIN {X 0,Y 457.754,Z 600.395,A -85,B 0,C 180,E1 -16098.526,E2 -16098.526} C_VEL
LIN {X 0,Y 457.807,Z 600.393,A -85,B 0,C 180,E1 -16102.085,E2 -16102.085} C_VEL
LIN {X 0,Y 457.872,Z 600.379,A -85,B 0,C 180,E1 -16104.733,E2 -16104.733} C_VEL
LIN {X 0,Y 457.744,Z 600.396,A -85,B 0,C 180,E1 -16107.369,E2 -16107.369} C_VEL
LIN {X 0,Y 457.949,Z 600.377,A -85,B 0,C 180,E1 -16110,E2 -16110} C_VEL
LIN {X 0,Y 457.904,Z 600.378,A -85,B 0,C 180,E1 -16114.386,E2 -16114.386} C_VEL
LIN {X 0,Y 457.818,Z 600.385,A -85,B 0,C 180,E1 -16117.03,E2 -16117.03} C_VEL
LIN {X 0,Y 457.723,Z 600.401,A -85,B 0,C 180,E1 -16119.691,E2 -16119.691} C_VEL
LIN {X 0,Y 457.731,Z 600.399,A -85,B 0,C 180,E1 -16122.371,E2 -16122.371} C_VEL
LIN {X 0,Y 457.739,Z 600.396,A -85,B 0,C 180,E1 -16125.414,E2 -16125.414} C_VEL
LIN {X 0,Y 457.643,Z 600.407,A -85,B 0,C 180,E1 -16128.748,E2 -16128.748} C_VEL
LIN {X 0,Y 457.633,Z 600.411,A -85,B 0,C 180,E1 -16131.551,E2 -16131.551} C_VEL
LIN {X 0,Y 457.581,Z 600.418,A -85,B 0,C 180,E1 -16134.412,E2 -16134.412} C_VEL
LIN {X 0,Y 457.618,Z 600.411,A -85,B 0,C 180,E1 -16137.407,E2 -16137.407} C_VEL
LIN {X 0,Y 457.632,Z 600.412,A -85,B 0,C 180,E1 -16140.337,E2 -16140.337} C_VEL
LIN {X 0,Y 457.616,Z 600.412,A -85,B 0,C 180,E1 -16142.219,E2 -16142.219} C_VEL
LIN {X 0,Y 456.993,Z 600.496,A -85,B 0,C 180,E1 -16142.954,E2 -16142.954} C_VEL
LIN {X 0,Y 454.157,Z 600.857,A -85,B 0,C 180,E1 -16144.147,E2 -16144.147} C_VEL
LIN {X 0,Y 451.731,Z 601.159,A -85,B 0,C 180,E1 -16145.11,E2 -16145.11} C_VEL
LIN {X 0,Y 450.688,Z 601.283,A -85,B 0,C 180,E1 -16145.854,E2 -16145.854} C_VEL
LIN {X 0,Y 450.604,Z 601.29,A -85,B 0,C 180,E1 -16146.106,E2 -16146.106} C_VEL
LIN {X 0,Y 450.57,Z 601.288,A -85,B 0,C 180,E1 -16148.988,E2 -16148.988} C_VEL
